C07289=1054.080,253.803,402.120,172.392,36.033,156.770
C07290=1054.086,254.052,402.091,172.395,36.036,156.771
C07291=1054.093,254.300,402.062,172.397,36.039,156.771
C07292=1054.100,254.548,402.034,172.400,36.043,156.772
C07293=1054.106,254.796,402.005,172.402,36.046,156.773
C07294=1054.112,255.044,401.976,172.404,36.050,156.774
C07295=1054.118,255.292,401.947,172.407,36.053,156.774
C07296=1054.125,255.540,401.918,172.410,36.056,156.775
C07297=1054.131,255.789,401.889,172.413,36.060,156.776
C07298=1054.138,256.037,401.859,172.415,36.063,156.777
C07299=1054.144,256.286,401.830,172.417,36.066,156.777
C07300=1054.150,256.534,401.801,172.420,36.070,156.778
C07301=1054.156,256.782,401.772,172.423,36.073,156.779
C07302=1054.163,257.030,401.743,172.425,36.077,156.779
C07303=1054.169,257.278,401.714,172.428,36.081,156.780
C07304=1054.176,257.527,401.685,172.430,36.083,156.781
C07305=1054.183,257.775,401.656,172.433,36.087,156.782
C07306=1054.189,258.023,401.627,172.436,36.091,156.782
C07307=1054.195,258.271,401.598,172.438,36.094,156.783
C07308=1054.201,258.519,401.569,172.441,36.097,156.784
C07309=1054.208,258.768,401.540,172.443,36.101,156.784
C07310=1054.215,259.016,401.511,172.445,36.104,156.785
C07311=1054.221,259.264,401.482,172.449,36.108,156.786
C07312=1054.227,259.512,401.453,172.451,36.111,156.787
C07313=1054.234,259.761,401.423,172.454,36.114,156.787
C07314=1054.241,260.009,401.393,172.456,36.118,156.788
C07315=1054.247,260.257,401.364,172.459,36.121,156.789
C07316=1054.253,260.505,401.335,172.462,36.124,156.789
C07317=1054.260,260.754,401.306,172.464,36.128,156.790
C07318=1054.266,261.002,401.277,172.467,36.131,156.791
C07319=1054.273,261.249,401.247,172.470,36.135,156.792
C07320=1054.279,261.498,401.218,172.472,36.138,156.792
C07321=1054.286,261.746,401.189,172.475,36.141,156.793
C07322=1054.292,261.995,401.160,172.477,36.145,156.794
C07323=1054.298,262.243,401.131,172.481,36.149,156.794
C07324=1054.304,262.456,401.105,172.483,36.151,156.795
C07325=1054.310,262.670,401.079,172.485,36.154,156.796
C07326=1054.316,262.884,401.055,172.487,36.157,156.796
C07327=1054.321,263.098,401.029,172.490,36.160,156.797
C07328=1054.327,263.312,401.003,172.491,36.163,156.798
C07329=1054.332,263.525,400.978,172.494,36.166,156.798
C07330=1054.337,263.740,400.952,172.496,36.169,156.799
C07331=1054.343,263.953,400.927,172.498,36.172,156.799
C07332=1054.351,264.254,400.890,172.502,36.176,156.800
C07333=1054.358,264.554,400.855,172.505,36.180,156.801
C07334=1054.366,264.855,400.819,172.509,36.185,156.802
C07335=1054.373,265.155,400.783,172.511,36.189,156.803
C07336=1054.380,265.403,400.753,172.515,36.192,156.804
C07337=1054.386,265.651,400.724,172.517,36.196,156.804
C07338=1054.392,265.899,400.694,172.519,36.199,156.805
C07339=1054.399,266.148,400.664,172.522,36.203,156.806
C07340=1054.406,266.396,400.635,172.525,36.206,156.807
C07341=1054.411,266.644,400.605,172.528,36.210,156.807
C07342=1054.418,266.892,400.575,172.530,36.213,156.808
C07343=1054.424,267.140,400.546,172.533,36.216,156.809
C07344=1054.431,267.389,400.515,172.536,36.220,156.810
C07345=1054.437,267.636,400.485,172.538,36.223,156.810
C07346=1054.444,267.885,400.456,172.542,36.227,156.811
C07347=1054.450,268.133,400.426,172.544,36.230,156.812
C07348=1054.456,268.381,400.396,172.546,36.234,156.813
C07349=1054.462,268.629,400.366,172.550,36.238,156.813
C07350=1054.469,268.877,400.336,172.552,36.241,156.814
C07351=1054.475,269.126,400.306,172.555,36.245,156.815
C07352=1054.482,269.374,400.276,172.558,36.248,156.816
C07353=1054.488,269.622,400.246,172.560,36.251,156.816
C07354=1054.494,269.869,400.216,172.563,36.255,156.817
C07355=1054.500,270.118,400.186,172.566,36.258,156.818
C07356=1054.507,270.366,400.156,172.569,36.262,156.818
C07357=1054.513,270.614,400.126,172.571,36.265,156.819
C07358=1054.520,270.862,400.096,172.575,36.269,156.820
C07359=1054.526,271.110,400.065,172.577,36.272,156.821
C07360=1054.533,271.359,400.036,172.579,36.276,156.821
C07361=1054.539,271.606,400.006,172.583,36.279,156.822
C07362=1054.546,271.855,399.976,172.585,36.283,156.823
C07363=1054.551,272.102,399.945,172.588,36.286,156.824
C07364=1054.559,272.351,399.915,172.591,36.290,156.825
C07365=1054.564,272.598,399.885,172.594,36.293,156.825
C07366=1054.571,272.847,399.854,172.597,36.297,156.826
C07367=1054.577,273.094,399.824,172.599,36.300,156.827
C07368=1054.584,273.343,399.794,172.602,36.304,156.828
C07369=1054.590,273.591,399.765,172.605,36.307,156.828
C07370=1054.597,273.840,399.734,172.608,36.311,156.829
C07371=1054.602,274.088,399.704,172.610,36.314,156.830
C07372=1054.609,274.336,399.673,172.613,36.318,156.831
C07373=1054.615,274.584,399.643,172.616,36.322,156.831
C07374=1054.622,274.831,399.612,172.619,36.324,156.832
C07375=1054.629,275.079,399.582,172.622,36.328,156.833
C07376=1054.635,275.327,399.551,172.624,36.331,156.833
C07377=1054.641,275.575,399.521,172.628,36.335,156.834
C07378=1054.647,275.824,399.490,172.630,36.339,156.835
C07379=1054.654,276.071,399.460,172.633,36.342,156.836
C07380=1054.660,276.314,399.431,172.636,36.346,156.836
C07381=1054.666,276.555,399.401,172.638,36.349,156.837
C07382=1054.672,276.798,399.371,172.642,36.353,156.838
C07383=1054.679,277.040,399.341,172.644,36.356,156.839
C07384=1054.685,277.282,399.311,172.647,36.360,156.839
C07385=1054.691,277.524,399.281,172.650,36.363,156.840
C07386=1054.697,277.766,399.252,172.652,36.367,156.841
C07387=1054.703,278.007,399.222,172.656,36.370,156.842
C07388=1054.710,278.256,399.192,172.658,36.373,156.842
C07389=1054.716,278.504,399.161,172.661,36.377,156.843
C07390=1054.723,278.751,399.130,172.664,36.381,156.844
C07391=1054.729,279.000,399.099,172.667,36.384,156.845
C07392=1054.735,279.248,399.069,172.670,36.388,156.846
C07393=1054.742,279.496,399.039,172.673,36.391,156.846
C07394=1054.749,279.744,399.007,172.676,36.395,156.847
C07395=1054.755,279.992,398.977,172.678,36.398,156.848
C07396=1054.761,280.240,398.946,172.682,36.402,156.849
C07397=1054.767,280.487,398.915,172.684,36.405,156.849
C07398=1054.774,280.736,398.884,172.688,36.409,156.850
C07399=1054.780,280.984,398.853,172.690,36.412,156.851
C07400=1054.786,281.232,398.822,172.693,36.416,156.852
C07401=1054.793,281.480,398.791,172.696,36.419,156.852
C07402=1054.799,281.728,398.760,172.699,36.423,156.853
C07403=1054.805,281.975,398.729,172.702,36.427,156.854
C07404=1054.812,282.224,398.699,172.704,36.430,156.855
C07405=1054.818,282.472,398.667,172.708,36.434,156.856
C07406=1054.824,282.720,398.637,172.710,36.437,156.856
C07407=1054.831,282.967,398.605,172.714,36.441,156.857
C07408=1054.837,283.216,398.575,172.716,36.444,156.858
C07409=1054.844,283.463,398.544,172.720,36.448,156.859
C07410=1054.850,283.712,398.513,172.722,36.452,156.859
C07411=1054.857,283.960,398.481,172.726,36.455,156.860
C07412=1054.863,284.207,398.451,172.728,36.459,156.861
C07413=1054.869,284.455,398.420,172.732,36.462,156.862
C07414=1054.876,284.703,398.388,172.734,36.466,156.862
C07415=1054.882,284.952,398.357,172.737,36.469,156.863
C07416=1054.889,285.199,398.326,172.740,36.473,156.864
C07417=1054.895,285.447,398.295,172.743,36.477,156.865
C07418=1054.902,285.695,398.264,172.746,36.481,156.866
C07419=1054.908,285.944,398.232,172.749,36.484,156.866
C07420=1054.914,286.191,398.201,172.753,36.488,156.867
C07421=1054.920,286.439,398.170,172.755,36.491,156.868
C07422=1054.927,286.687,398.139,172.759,36.495,156.869
C07423=1054.934,286.935,398.108,172.761,36.498,156.869
C07424=1054.940,287.183,398.076,172.765,36.502,156.870
C07425=1054.946,287.431,398.046,172.767,36.506,156.871
C07426=1054.953,287.679,398.014,172.771,36.509,156.872
C07427=1054.960,287.927,397.983,172.773,36.513,156.873
C07428=1054.966,288.175,397.951,172.776,36.516,156.873
C07429=1054.973,288.422,397.920,172.780,36.520,156.874
C07430=1054.978,288.670,397.888,172.782,36.524,156.875
C07431=1054.985,288.918,397.857,172.786,36.527,156.876
C07432=1054.992,289.166,397.826,172.788,36.531,156.877
C07433=1054.998,289.414,397.795,172.792,36.534,156.877
C07434=1055.004,289.662,397.763,172.794,36.538,156.878
C07435=1055.011,289.910,397.731,172.798,36.542,156.879
C07436=1055.017,290.158,397.700,172.801,36.545,156.880
C07437=1055.024,290.405,397.668,172.804,36.549,156.881
C07438=1055.030,290.652,397.637,172.807,36.553,156.881
C07439=1055.037,290.900,397.606,172.810,36.556,156.882
C07440=1055.042,291.147,397.574,172.813,36.560,156.883
C07441=1055.049,291.395,397.542,172.817,36.563,156.884
C07442=1055.056,291.643,397.510,172.819,36.567,156.885
C07443=1055.062,291.890,397.479,172.823,36.571,156.885
C07444=1055.068,292.138,397.447,172.825,36.574,156.886
C07445=1055.075,292.386,397.416,172.829,36.578,156.887
C07446=1055.082,292.634,397.384,172.832,36.582,156.888
C07447=1055.088,292.882,397.352,172.835,36.585,156.889
C07448=1055.095,293.129,397.320,172.838,36.589,156.889
C07449=1055.101,293.377,397.289,172.842,36.593,156.890
C07450=1055.107,293.625,397.257,172.844,36.596,156.891
C07451=1055.114,293.873,397.225,172.848,36.600,156.892
C07452=1055.120,294.121,397.194,172.850,36.604,156.893
C07453=1055.127,294.368,397.162,172.854,36.607,156.893
C07454=1055.133,294.616,397.130,172.857,36.611,156.894
C07455=1055.139,294.864,397.098,172.860,36.615,156.895
C07456=1055.146,295.112,397.067,172.863,36.618,156.896
C07457=1055.152,295.360,397.034,172.867,36.622,156.897
C07458=1055.159,295.608,397.002,172.869,36.626,156.898
C07459=1055.165,295.856,396.970,172.872,36.629,156.898
C07460=1055.172,296.103,396.938,172.876,36.633,156.899
C07461=1055.178,296.351,396.906,172.879,36.637,156.900
C07462=1055.185,296.599,396.874,172.882,36.640,156.901
C07463=1055.191,296.847,396.842,172.886,36.644,156.902
C07464=1055.197,297.095,396.810,172.888,36.648,156.903
C07465=1055.204,297.342,396.778,172.892,36.652,156.903
C07466=1055.210,297.591,396.746,172.895,36.656,156.904
C07467=1055.216,297.838,396.713,172.898,36.659,156.905
C07468=1055.222,298.086,396.681,172.901,36.663,156.906
C07469=1055.229,298.334,396.648,172.905,36.667,156.907
C07470=1055.236,298.581,396.616,172.907,36.671,156.908
C07471=1055.242,298.829,396.584,172.911,36.674,156.908
C07472=1055.248,299.077,396.551,172.914,36.678,156.909
C07473=1055.254,299.325,396.519,172.917,36.682,156.910
C07474=1055.261,299.573,396.487,172.920,36.686,156.911
C07475=1055.267,299.820,396.455,172.924,36.690,156.912
C07476=1055.273,300.068,396.423,172.926,36.693,156.913
C07477=1055.280,300.316,396.390,172.930,36.697,156.913
C07478=1055.286,300.564,396.357,172.933,36.701,156.914
C07479=1055.293,300.811,396.326,172.937,36.705,156.915
C07480=1055.299,301.059,396.293,172.939,36.709,156.916
C07481=1055.305,301.307,396.260,172.943,36.712,156.917
C07482=1055.311,301.555,396.228,172.946,36.717,156.918
C07483=1055.317,301.802,396.195,172.950,36.720,156.918
C07484=1055.324,302.050,396.163,172.953,36.724,156.919
C07485=1055.331,302.298,396.130,172.956,36.728,156.920
C07486=1055.338,302.546,396.097,172.960,36.731,156.921
C07487=1055.344,302.794,396.065,172.963,36.736,156.922
C07488=1055.350,303.041,396.033,172.966,36.739,156.923
C07489=1055.356,303.289,396.000,172.969,36.743,156.924
C07490=1055.363,303.537,395.967,172.973,36.747,156.924
C07491=1055.370,303.784,395.935,172.976,36.751,156.925
C07492=1055.376,304.047,395.900,172.979,36.755,156.926
C07493=1055.383,304.310,395.866,172.982,36.759,156.927
C07494=1055.390,304.573,395.831,172.986,36.763,156.928
C07495=1055.396,304.836,395.796,172.990,36.767,156.929
C07496=1055.404,305.084,395.764,172.993,36.771,156.930
C07497=1055.410,305.332,395.731,172.997,36.775,156.931
C07498=1055.417,305.580,395.698,173.000,36.778,156.931
C07499=1055.423,305.827,395.666,173.004,36.782,156.932
C07500=1055.429,306.075,395.633,173.006,36.786,156.933
C07501=1055.436,306.323,395.600,173.010,36.790,156.934
C07502=1055.442,306.571,395.567,173.013,36.794,156.935
C07503=1055.449,306.818,395.534,173.017,36.798,156.936
C07504=1055.456,307.065,395.501,173.020,36.801,156.937
C07505=1055.463,307.313,395.468,173.023,36.805,156.938
C07506=1055.469,307.561,395.436,173.027,36.809,156.938
C07507=1055.475,307.808,395.403,173.030,36.813,156.939
C07508=1055.482,308.057,395.370,173.034,36.817,156.940
C07509=1055.489,308.304,395.337,173.037,36.821,156.941
C07510=1055.495,308.552,395.304,173.041,36.825,156.942
C07511=1055.502,308.800,395.271,173.044,36.828,156.943
C07512=1055.508,309.047,395.238,173.047,36.832,156.944
C07513=1055.515,309.294,395.205,173.051,36.836,156.945
C07514=1055.522,309.543,395.172,173.054,36.840,156.945
C07515=1055.529,309.790,395.140,173.058,36.844,156.946
C07516=1055.535,310.037,395.106,173.061,36.848,156.947
C07517=1055.542,310.286,395.073,173.065,36.852,156.948
C07518=1055.548,310.533,395.040,173.068,36.855,156.949
C07519=1055.555,310.781,395.007,173.071,36.859,156.950
C07520=1055.562,311.028,394.974,173.074,36.863,156.951
C07521=1055.569,311.277,394.941,173.078,36.867,156.952
C07522=1055.575,311.524,394.908,173.082,36.871,156.952
C07523=1055.582,311.771,394.874,173.085,36.875,156.953
C07524=1055.589,312.020,394.841,173.089,36.879,156.954
C07525=1055.595,312.267,394.808,173.092,36.883,156.955
C07526=1055.602,312.515,394.775,173.096,36.886,156.956
C07527=1055.608,312.762,394.742,173.099,36.890,156.957
C07528=1055.616,313.010,394.708,173.103,36.894,156.958
C07529=1055.622,313.258,394.675,173.107,36.898,156.959
C07530=1055.629,313.505,394.642,173.109,36.902,156.959
C07531=1055.635,313.753,394.609,173.113,36.906,156.960
C07532=1055.642,314.001,394.574,173.116,36.910,156.961
C07533=1055.648,314.248,394.541,173.120,36.914,156.962
C07534=1055.655,314.497,394.507,173.124,36.918,156.963
C07535=1055.661,314.743,394.474,173.127,36.922,156.964
C07536=1055.667,314.991,394.440,173.131,36.926,156.965
C07537=1055.674,315.239,394.407,173.134,36.930,156.966
C07538=1055.681,315.486,394.373,173.138,36.934,156.967
C07539=1055.687,315.734,394.339,173.142,36.939,156.968
C07540=1055.693,315.982,394.306,173.144,36.943,156.969
C07541=1055.700,316.230,394.272,173.148,36.947,156.970
C07542=1055.706,316.477,394.238,173.151,36.951,156.970
C07543=1055.713,316.725,394.204,173.155,36.955,156.971
C07544=1055.719,316.972,394.171,173.159,36.959,156.972
C07545=1055.726,317.220,394.137,173.162,36.963,156.973
C07546=1055.732,317.467,394.103,173.166,36.967,156.974
C07547=1055.739,317.715,394.069,173.170,36.971,156.975
C07548=1055.745,317.982,394.032,173.173,36.975,156.976
C07549=1055.752,318.249,393.996,173.177,36.980,156.977
C07550=1055.759,318.516,393.959,173.182,36.984,156.978
C07551=1055.767,318.784,393.922,173.185,36.989,156.979
C07552=1055.773,319.031,393.889,173.189,36.993,156.980
C07553=1055.780,319.279,393.854,173.192,36.997,156.981
C07554=1055.786,319.527,393.821,173.196,37.001,156.982
C07555=1055.792,319.774,393.787,173.200,37.005,156.983
C07556=1055.800,320.022,393.753,173.203,37.009,156.984
C07557=1055.805,320.269,393.719,173.207,37.013,156.985
C07558=1055.813,320.517,393.685,173.211,37.017,156.986
C07559=1055.819,320.764,393.650,173.214,37.021,156.987
C07560=1055.826,321.011,393.617,173.218,37.026,156.988
C07561=1055.832,321.259,393.582,173.221,37.030,156.989
C07562=1055.839,321.507,393.548,173.225,37.034,156.990
C07563=1055.845,321.754,393.514,173.229,37.038,156.990
C07564=1055.852,322.002,393.480,173.232,37.042,156.992
C07565=1055.859,322.250,393.446,173.236,37.046,156.992
C07566=1055.866,322.498,393.412,173.240,37.050,156.993
C07567=1055.872,322.745,393.378,173.243,37.054,156.994
C07568=1055.879,322.992,393.343,173.247,37.059,156.995
C07569=1055.885,323.240,393.309,173.251,37.063,156.996
C07570=1055.893,323.488,393.275,173.254,37.067,156.997
C07571=1055.898,323.735,393.241,173.258,37.071,156.998
C07572=1055.906,323.983,393.207,173.262,37.075,156.999
C07573=1055.912,324.230,393.172,173.265,37.079,157.000
C07574=1055.919,324.478,393.138,173.269,37.084,157.001
C07575=1055.926,324.726,393.104,173.272,37.088,157.002
C07576=1055.932,324.972,393.069,173.276,37.092,157.003
C07577=1055.939,325.220,393.035,173.280,37.096,157.004
C07578=1055.946,325.468,393.001,173.284,37.100,157.005
C07579=1055.953,325.715,392.966,173.288,37.105,157.006
C07580=1055.960,325.963,392.932,173.292,37.109,157.007
C07581=1055.966,326.211,392.897,173.295,37.113,157.008
C07582=1055.973,326.458,392.862,173.299,37.117,157.009
C07583=1055.980,326.705,392.829,173.303,37.121,157.010
C07584=1055.987,326.953,392.794,173.306,37.126,157.011
C07585=1055.993,327.201,392.759,173.310,37.130,157.012
C07586=1056.000,327.448,392.725,173.314,37.134,157.013
C07587=1056.007,327.696,392.690,173.318,37.138,157.014
C07588=1056.014,327.943,392.656,173.322,37.142,157.015
C07589=1056.021,328.191,392.621,173.326,37.147,157.016
C07590=1056.028,328.438,392.586,173.329,37.151,157.017
C07591=1056.035,328.686,392.552,173.333,37.155,157.018
C07592=1056.042,328.933,392.517,173.337,37.159,157.019
C07593=1056.048,329.181,392.482,173.341,37.164,157.020
C07594=1056.056,329.428,392.448,173.345,37.168,157.021
C07595=1056.062,329.676,392.413,173.349,37.172,157.022
C07596=1056.069,329.924,392.379,173.353,37.176,157.023
C07597=1056.076,330.171,392.343,173.356,37.181,157.024
C07598=1056.082,330.418,392.308,173.360,37.185,157.025
C07599=1056.089,330.666,392.273,173.364,37.189,157.026
C07600=1056.096,330.914,392.239,173.368,37.194,157.027
C07601=1056.102,331.161,392.204,173.372,37.198,157.028
C07602=1056.109,331.408,392.169,173.376,37.203,157.029
C07603=1056.116,331.656,392.133,173.379,37.207,157.030
C07604=1056.123,331.918,392.097,173.383,37.212,157.031
C07605=1056.130,332.179,392.059,173.388,37.216,157.032
C07606=1056.137,332.441,392.023,173.392,37.221,157.033
C07607=1056.144,332.703,391.985,173.397,37.225,157.034
C07608=1056.151,332.950,391.950,173.400,37.230,157.035
C07609=1056.158,333.198,391.914,173.404,37.234,157.036
C07610=1056.165,333.445,391.879,173.408,37.239,157.037
C07611=1056.172,333.692,391.844,173.411,37.243,157.038
C07612=1056.178,333.940,391.809,173.416,37.248,157.039
C07613=1056.185,334.187,391.774,173.420,37.252,157.040
C07614=1056.192,334.435,391.739,173.424,37.256,157.041
C07615=1056.199,334.682,391.704,173.427,37.261,157.042
C07616=1056.205,334.929,391.669,173.432,37.265,157.043
C07617=1056.213,335.177,391.633,173.436,37.270,157.045
C07618=1056.219,335.425,391.597,173.440,37.274,157.046
C07619=1056.226,335.672,391.562,173.443,37.279,157.047
C07620=1056.233,335.919,391.526,173.448,37.283,157.048
C07621=1056.239,336.167,391.491,173.452,37.288,157.049
C07622=1056.246,336.414,391.456,173.456,37.292,157.050
C07623=1056.254,336.662,391.421,173.459,37.297,157.051
C07624=1056.260,336.909,391.385,173.464,37.301,157.052
C07625=1056.267,337.156,391.349,173.468,37.306,157.053
C07626=1056.273,337.404,391.314,173.472,37.310,157.054
C07627=1056.280,337.651,391.279,173.475,37.315,157.055
C07628=1056.287,337.898,391.242,173.480,37.319,157.056
C07629=1056.294,338.146,391.207,173.484,37.324,157.057
C07630=1056.301,338.393,391.171,173.488,37.329,157.058
C07631=1056.307,338.641,391.135,173.491,37.333,157.060
C07632=1056.314,338.888,391.100,173.496,37.338,157.061
C07633=1056.321,339.135,391.064,173.500,37.342,157.062
C07634=1056.327,339.383,391.028,173.504,37.347,157.063
C07635=1056.335,339.630,390.992,173.509,37.352,157.064
C07636=1056.341,339.877,390.957,173.512,37.356,157.065
C07637=1056.348,340.125,390.920,173.516,37.361,157.066
C07638=1056.355,340.372,390.885,173.521,37.365,157.067
C07639=1056.362,340.619,390.849,173.525,37.370,157.068
C07640=1056.368,340.867,390.814,173.528,37.375,157.069
C07641=1056.376,341.114,390.777,173.533,37.379,157.070
C07642=1056.382,341.361,390.741,173.537,37.384,157.072
C07643=1056.389,341.609,390.706,173.541,37.389,157.073
C07644=1056.397,341.856,390.670,173.546,37.393,157.074
C07645=1056.403,342.103,390.633,173.549,37.398,157.075
C07646=1056.410,342.351,390.598,173.553,37.403,157.076
C07647=1056.417,342.598,390.562,173.558,37.407,157.077
C07648=1056.424,342.845,390.525,173.562,37.412,157.078
C07649=1056.431,343.093,390.490,173.567,37.417,157.079
C07650=1056.437,343.340,390.453,173.570,37.421,157.081
C07651=1056.444,343.587,390.417,173.574,37.426,157.082
C07652=1056.451,343.835,390.381,173.579,37.431,157.083
C07653=1056.458,344.082,390.344,173.583,37.436,157.084
C07654=1056.465,344.329,390.308,173.587,37.440,157.085
C07655=1056.472,344.576,390.272,173.592,37.445,157.086
C07656=1056.479,344.824,390.236,173.595,37.450,157.087
C07657=1056.485,345.071,390.200,173.600,37.455,157.089
C07658=1056.492,345.318,390.163,173.604,37.459,157.090
C07659=1056.499,345.566,390.127,173.608,37.464,157.091
C07660=1056.506,345.823,390.089,173.613,37.469,157.092
C07661=1056.514,346.080,390.051,173.618,37.474,157.093
C07662=1056.520,346.338,390.013,173.622,37.479,157.094
C07663=1056.528,346.596,389.975,173.626,37.484,157.096
C07664=1056.535,346.843,389.939,173.630,37.489,157.097
C07665=1056.542,347.091,389.902,173.635,37.494,157.098
C07666=1056.548,347.337,389.865,173.639,37.499,157.099
C07667=1056.556,347.584,389.829,173.644,37.504,157.100
C07668=1056.563,347.832,389.792,173.648,37.508,157.101
C07669=1056.569,348.079,389.756,173.652,37.513,157.103
C07670=1056.577,348.327,389.719,173.656,37.518,157.104
C07671=1056.584,348.573,389.682,173.660,37.523,157.105
C07672=1056.590,348.821,389.645,173.665,37.528,157.106
C07673=1056.597,349.068,389.609,173.669,37.533,157.107
C07674=1056.605,349.315,389.573,173.674,37.538,157.109
C07675=1056.611,349.562,389.536,173.678,37.543,157.110
C07676=1056.618,349.810,389.499,173.683,37.548,157.111
C07677=1056.625,350.057,389.462,173.687,37.553,157.112
C07678=1056.632,350.303,389.425,173.692,37.558,157.113
C07679=1056.639,350.551,389.389,173.695,37.563,157.115
C07680=1056.647,350.798,389.351,173.700,37.568,157.116
C07681=1056.653,351.045,389.315,173.704,37.572,157.117
C07682=1056.660,351.293,389.278,173.709,37.577,157.118
C07683=1056.668,351.540,389.241,173.713,37.583,157.119
C07684=1056.674,351.787,389.204,173.718,37.588,157.121
C07685=1056.681,352.034,389.167,173.723,37.593,157.122
C07686=1056.689,352.281,389.129,173.727,37.598,157.123
C07687=1056.695,352.528,389.093,173.732,37.603,157.124
C07688=1056.702,352.776,389.055,173.736,37.608,157.126
C07689=1056.709,353.023,389.019,173.740,37.613,157.127
C07690=1056.716,353.270,388.981,173.744,37.618,157.128
C07691=1056.723,353.517,388.944,173.749,37.623,157.129
C07692=1056.730,353.764,388.906,173.753,37.628,157.131
C07693=1056.737,354.012,388.869,173.758,37.633,157.132
C07694=1056.744,354.258,388.832,173.763,37.638,157.133
C07695=1056.751,354.505,388.795,173.767,37.643,157.134
C07696=1056.758,354.752,388.757,173.772,37.649,157.136
C07697=1056.765,355.000,388.720,173.776,37.654,157.137
C07698=1056.772,355.247,388.683,173.781,37.659,157.138
C07699=1056.779,355.494,388.646,173.786,37.664,157.139
C07700=1056.786,355.741,388.608,173.790,37.669,157.141
C07701=1056.794,355.988,388.571,173.795,37.674,157.142
C07702=1056.801,356.235,388.533,173.799,37.680,157.143
C07703=1056.808,356.482,388.496,173.804,37.685,157.144
C07704=1056.815,356.729,388.459,173.809,37.689,157.146
C07705=1056.822,356.976,388.421,173.813,37.695,157.147
C07706=1056.829,357.223,388.383,173.818,37.700,157.148
C07707=1056.837,357.470,388.346,173.823,37.705,157.149
C07708=1056.844,357.717,388.308,173.827,37.710,157.151
C07709=1056.850,357.965,388.270,173.831,37.715,157.152
C07710=1056.858,358.212,388.233,173.837,37.721,157.153
C07711=1056.865,358.459,388.195,173.841,37.726,157.155
C07712=1056.872,358.706,388.158,173.845,37.731,157.156
C07713=1056.879,358.953,388.121,173.851,37.737,157.157
C07714=1056.885,359.200,388.082,173.854,37.742,157.158
C07715=1056.893,359.447,388.044,173.860,37.747,157.160
C07716=1056.900,359.709,388.004,173.865,37.753,157.161
C07717=1056.908,359.971,387.964,173.870,37.759,157.163
C07718=1056.916,360.234,387.924,173.875,37.765,157.164
C07719=1056.923,360.497,387.883,173.880,37.770,157.165
C07720=1056.931,360.744,387.845,173.884,37.776,157.167
C07721=1056.938,360.991,387.808,173.889,37.781,157.168
C07722=1056.945,361.237,387.769,173.894,37.787,157.169
C07723=1056.952,361.485,387.731,173.899,37.791,157.171
C07724=1056.959,361.732,387.694,173.903,37.797,157.172
C07725=1056.967,361.979,387.655,173.908,37.802,157.173
C07726=1056.974,362.226,387.618,173.913,37.808,157.175
C07727=1056.981,362.473,387.579,173.918,37.813,157.176
C07728=1056.988,362.720,387.542,173.922,37.819,157.178
C07729=1056.996,362.966,387.503,173.927,37.824,157.179
C07730=1057.002,363.213,387.465,173.932,37.830,157.180
C07731=1057.010,363.460,387.427,173.937,37.835,157.182
C07732=1057.017,363.707,387.389,173.941,37.841,157.183
C07733=1057.024,363.954,387.351,173.946,37.846,157.184
C07734=1057.030,364.201,387.312,173.952,37.852,157.186
C07735=1057.038,364.447,387.274,173.957,37.857,157.187
C07736=1057.045,364.695,387.234,173.961,37.863,157.188
C07737=1057.053,364.942,387.197,173.966,37.868,157.190
C07738=1057.059,365.189,387.158,173.971,37.874,157.191
C07739=1057.067,365.435,387.120,173.976,37.880,157.193
C07740=1057.074,365.682,387.081,173.981,37.885,157.194
C07741=1057.081,365.929,387.043,173.986,37.891,157.195
C07742=1057.088,366.176,387.004,173.990,37.897,157.197
C07743=1057.095,366.424,386.965,173.995,37.902,157.198
C07744=1057.103,366.670,386.927,174.000,37.908,157.200
C07745=1057.110,366.917,386.888,174.006,37.914,157.201
C07746=1057.117,367.164,386.850,174.011,37.919,157.203
C07747=1057.124,367.410,386.811,174.016,37.925,157.204
C07748=1057.131,367.658,386.772,174.020,37.931,157.205
C07749=1057.139,367.904,386.734,174.025,37.936,157.207
C07750=1057.146,368.151,386.695,174.030,37.942,157.208
C07751=1057.154,368.398,386.656,174.035,37.948,157.210
C07752=1057.161,368.645,386.617,174.041,37.954,157.211
C07753=1057.168,368.892,386.578,174.046,37.959,157.213
C07754=1057.175,369.138,386.540,174.051,37.965,157.214
C07755=1057.183,369.386,386.500,174.056,37.971,157.216
C07756=1057.190,369.632,386.462,174.060,37.977,157.217
C07757=1057.198,369.878,386.423,174.065,37.982,157.218
C07758=1057.205,370.126,386.383,174.070,37.988,157.220
C07759=1057.212,370.372,386.345,174.076,37.994,157.221
C07760=1057.220,370.620,386.306,174.081,38.000,157.223
C07761=1057.227,370.866,386.266,174.086,38.006,157.224
C07762=1057.235,371.113,386.228,174.091,38.012,157.226
C07763=1057.242,371.359,386.188,174.096,38.017,157.227
C07764=1057.249,371.606,386.149,174.101,38.023,157.229
C07765=1057.257,371.854,386.111,174.107,38.029,157.230
C07766=1057.264,372.100,386.071,174.112,38.035,157.232
C07767=1057.272,372.347,386.032,174.117,38.041,157.233
C07768=1057.279,372.593,385.993,174.122,38.047,157.235
C07769=1057.286,372.840,385.954,174.128,38.053,157.236
C07770=1057.293,373.087,385.914,174.133,38.059,157.238
C07771=1057.301,373.333,385.874,174.138,38.065,157.239
C07772=1057.309,373.615,385.830,174.143,38.072,157.241
C07773=1057.317,373.896,385.785,174.150,38.079,157.243
C07774=1057.327,374.177,385.740,174.155,38.086,157.245
C07775=1057.334,374.458,385.695,174.162,38.092,157.246
C07776=1057.342,374.705,385.655,174.167,38.099,157.248
C07777=1057.349,374.951,385.615,174.172,38.105,157.249
C07778=1057.356,375.198,385.576,174.177,38.111,157.251
C07779=1057.364,375.444,385.536,174.183,38.117,157.253
C07780=1057.371,375.691,385.497,174.188,38.123,157.254
C07781=1057.378,375.938,385.457,174.193,38.129,157.256
C07782=1057.386,376.185,385.417,174.198,38.135,157.257
C07783=1057.394,376.431,385.377,174.204,38.141,157.259
C07784=1057.401,376.678,385.338,174.209,38.148,157.260
C07785=1057.408,376.925,385.298,174.214,38.154,157.262
C07786=1057.416,377.172,385.258,174.221,38.160,157.264
C07787=1057.423,377.418,385.218,174.226,38.166,157.265
C07788=1057.431,377.665,385.179,174.231,38.172,157.267
C07789=1057.439,377.912,385.139,174.237,38.179,157.268
C07790=1057.446,378.158,385.099,174.242,38.185,157.270
C07791=1057.454,378.404,385.058,174.247,38.191,157.272
C07792=1057.462,378.651,385.019,174.253,38.198,157.273
C07793=1057.469,378.897,384.979,174.258,38.204,157.275
C07794=1057.476,379.144,384.939,174.263,38.210,157.276
C07795=1057.484,379.391,384.899,174.269,38.216,157.278
C07796=1057.492,379.637,384.858,174.275,38.222,157.280
C07797=1057.499,379.883,384.819,174.280,38.229,157.281
C07798=1057.507,380.130,384.779,174.285,38.235,157.283
C07799=1057.515,380.377,384.739,174.291,38.241,157.284
C07800=1057.523,380.624,384.698,174.296,38.248,157.286
C07801=1057.530,380.870,384.659,174.303,38.254,157.288
C07802=1057.537,381.116,384.618,174.308,38.261,157.290
C07803=1057.545,381.363,384.578,174.313,38.267,157.291
C07804=1057.553,381.609,384.537,174.319,38.274,157.293
C07805=1057.560,381.857,384.497,174.324,38.280,157.295
C07806=1057.568,382.103,384.456,174.331,38.287,157.296
C07807=1057.575,382.349,384.415,174.336,38.293,157.298
C07808=1057.582,382.596,384.375,174.341,38.300,157.300
C07809=1057.590,382.842,384.335,174.347,38.306,157.301
C07810=1057.598,383.089,384.293,174.352,38.313,157.303
C07811=1057.605,383.336,384.253,174.359,38.320,157.305
C07812=1057.613,383.582,384.213,174.364,38.326,157.306
C07813=1057.621,383.828,384.172,174.370,38.333,157.308
C07814=1057.629,384.075,384.131,174.375,38.340,157.310
C07815=1057.636,384.322,384.090,174.381,38.346,157.312
C07816=1057.644,384.568,384.050,174.387,38.353,157.313
C07817=1057.651,384.814,384.009,174.392,38.360,157.315
C07818=1057.658,385.060,383.968,174.399,38.366,157.317
C07819=1057.667,385.307,383.927,174.404,38.373,157.319
C07820=1057.674,385.553,383.887,174.410,38.379,157.320
C07821=1057.682,385.800,383.845,174.416,38.386,157.322
C07822=1057.690,386.047,383.805,174.422,38.393,157.324
C07823=1057.698,386.293,383.764,174.427,38.400,157.326
C07824=1057.706,386.539,383.723,174.434,38.406,157.327
C07825=1057.713,386.786,383.682,174.439,38.413,157.329
C07826=1057.721,387.032,383.641,174.445,38.420,157.331
C07827=1057.729,387.279,383.600,174.451,38.427,157.333
C07828=1057.738,387.591,383.548,174.458,38.435,157.335
C07829=1057.749,387.903,383.496,174.466,38.444,157.337
C07830=1057.759,388.216,383.444,174.473,38.453,157.340
C07831=1057.768,388.529,383.392,174.481,38.462,157.342
C07832=1057.777,388.775,383.350,174.487,38.469,157.344
C07833=1057.784,389.021,383.309,174.493,38.475,157.345
C07834=1057.792,389.267,383.268,174.499,38.482,157.347
C07835=1057.801,389.514,383.227,174.505,38.489,157.349
C07836=1057.808,389.760,383.185,174.511,38.496,157.351
C07837=1057.816,390.006,383.143,174.516,38.503,157.353
C07838=1057.824,390.253,383.103,174.523,38.510,157.355
C07839=1057.832,390.499,383.060,174.529,38.517,157.356
C07840=1057.839,390.746,383.019,174.535,38.524,157.358
C07841=1057.848,390.992,382.978,174.541,38.531,157.360
C07842=1057.855,391.238,382.937,174.547,38.539,157.362
C07843=1057.863,391.485,382.894,174.553,38.546,157.364
C07844=1057.871,391.730,382.853,174.560,38.552,157.366
C07845=1057.879,391.977,382.812,174.565,38.560,157.368
C07846=1057.887,392.224,382.769,174.572,38.567,157.370
C07847=1057.894,392.470,382.728,174.578,38.574,157.372
C07848=1057.903,392.715,382.686,174.584,38.581,157.373
C07849=1057.911,392.962,382.644,174.590,38.589,157.375
C07850=1057.918,393.209,382.603,174.597,38.596,157.377
C07851=1057.926,393.455,382.560,174.602,38.603,157.379
C07852=1057.934,393.701,382.518,174.609,38.610,157.381
C07853=1057.942,393.947,382.476,174.615,38.618,157.383
C07854=1057.951,394.194,382.435,174.621,38.625,157.385
C07855=1057.958,394.440,382.393,174.628,38.632,157.387
C07856=1057.966,394.686,382.350,174.634,38.640,157.389
C07857=1057.974,394.932,382.308,174.641,38.647,157.391
C07858=1057.982,395.179,382.266,174.646,38.654,157.393
C07859=1057.990,395.424,382.224,174.653,38.662,157.395
C07860=1057.998,395.671,382.181,174.660,38.669,157.397
C07861=1058.006,395.917,382.139,174.666,38.677,157.399
C07862=1058.014,396.164,382.097,174.672,38.684,157.401
C07863=1058.022,396.410,382.055,174.679,38.691,157.403
C07864=1058.030,396.656,382.012,174.685,38.699,157.405
C07865=1058.038,396.902,381.970,174.692,38.706,157.407
C07866=1058.047,397.148,381.928,174.697,38.714,157.409
C07867=1058.054,397.394,381.885,174.704,38.722,157.411
C07868=1058.063,397.641,381.842,174.711,38.729,157.413
C07869=1058.070,397.887,381.800,174.717,38.737,157.415
C07870=1058.079,398.133,381.757,174.724,38.745,157.417
C07871=1058.087,398.380,381.715,174.730,38.752,157.419
C07872=1058.095,398.625,381.672,174.737,38.760,157.421
C07873=1058.103,398.871,381.629,174.743,38.767,157.423
C07874=1058.112,399.118,381.587,174.750,38.775,157.425
C07875=1058.119,399.363,381.544,174.757,38.783,157.428
C07876=1058.127,399.610,381.502,174.763,38.791,157.430
C07877=1058.135,399.856,381.459,174.770,38.799,157.432
C07878=1058.144,400.102,381.415,174.777,38.807,157.434
C07879=1058.152,400.348,381.372,174.783,38.814,157.436
C07880=1058.160,400.594,381.331,174.790,38.822,157.438
C07881=1058.168,400.840,381.287,174.796,38.830,157.440
C07882=1058.176,401.087,381.244,174.803,38.838,157.442
C07883=1058.185,401.333,381.201,174.810,38.846,157.445
C07884=1058.196,401.663,381.144,174.819,38.856,157.447
C07885=1058.207,401.992,381.086,174.828,38.867,157.450
C07886=1058.218,402.323,381.028,174.837,38.877,157.453
C07887=1058.229,402.652,380.970,174.846,38.888,157.456
C07888=1058.237,402.898,380.926,174.853,38.896,157.458
C07889=1058.245,403.144,380.883,174.860,38.904,157.460
C07890=1058.254,403.390,380.840,174.866,38.912,157.463
C07891=1058.262,403.637,380.797,174.873,38.920,157.465
C07892=1058.270,403.882,380.753,174.881,38.929,157.467
C07893=1058.279,404.128,380.710,174.887,38.936,157.469
C07894=1058.287,404.374,380.666,174.895,38.945,157.472
C07895=1058.295,404.621,380.623,174.902,38.953,157.474
C07896=1058.304,404.867,380.579,174.909,38.961,157.476
C07897=1058.312,405.113,380.536,174.916,38.969,157.478
C07898=1058.320,405.359,380.491,174.923,38.977,157.481
C07899=1058.329,405.605,380.448,174.930,38.986,157.483
C07900=1058.337,405.851,380.405,174.937,38.994,157.485
C07901=1058.345,406.097,380.361,174.944,39.003,157.487
C07902=1058.354,406.342,380.317,174.951,39.011,157.490
C07903=1058.361,406.589,380.273,174.958,39.019,157.492
C07904=1058.371,406.835,380.229,174.965,39.027,157.494
C07905=1058.378,407.081,380.185,174.972,39.036,157.497
C07906=1058.387,407.327,380.141,174.980,39.045,157.499
C07907=1058.395,407.572,380.097,174.987,39.053,157.501
C07908=1058.404,407.819,380.052,174.994,39.061,157.504
C07909=1058.413,408.065,380.009,175.001,39.070,157.506
C07910=1058.421,408.311,379.965,175.008,39.078,157.508
C07911=1058.429,408.556,379.921,175.016,39.087,157.511
C07912=1058.438,408.803,379.877,175.023,39.095,157.513
C07913=1058.446,409.048,379.832,175.030,39.104,157.515
C07914=1058.454,409.294,379.788,175.037,39.113,157.518
C07915=1058.464,409.540,379.744,175.045,39.121,157.520
C07916=1058.472,409.786,379.700,175.053,39.130,157.523
C07917=1058.480,410.032,379.655,175.060,39.139,157.525
C07918=1058.489,410.278,379.611,175.067,39.147,157.527
C07919=1058.498,410.524,379.566,175.074,39.156,157.530
C07920=1058.506,410.770,379.522,175.083,39.165,157.532
C07921=1058.514,411.015,379.477,175.090,39.173,157.535
C07922=1058.524,411.261,379.433,175.097,39.182,157.537
C07923=1058.532,411.508,379.388,175.105,39.191,157.540
C07924=1058.540,411.753,379.344,175.112,39.200,157.542
C07925=1058.550,411.999,379.299,175.120,39.209,157.545
C07926=1058.558,412.245,379.255,175.128,39.218,157.547
C07927=1058.567,412.491,379.210,175.135,39.227,157.550
C07928=1058.575,412.736,379.165,175.143,39.235,157.552
C07929=1058.585,412.982,379.121,175.151,39.244,157.555
C07930=1058.594,413.228,379.075,175.158,39.254,157.557
C07931=1058.602,413.474,379.031,175.166,39.262,157.560
C07932=1058.611,413.720,378.986,175.174,39.271,157.562
C07933=1058.619,413.966,378.941,175.181,39.281,157.565
C07934=1058.628,414.212,378.896,175.190,39.289,157.567
C07935=1058.637,414.457,378.850,175.197,39.299,157.570
C07936=1058.646,414.703,378.805,175.205,39.308,157.573
C07937=1058.655,414.949,378.760,175.213,39.317,157.575
C07938=1058.663,415.195,378.715,175.221,39.326,157.578
C07939=1058.672,415.440,378.670,175.229,39.336,157.580
C07940=1058.679,415.655,378.630,175.235,39.344,157.583
C07941=1058.687,415.870,378.591,175.242,39.352,157.585
C07942=1058.696,416.085,378.551,175.250,39.360,157.587
C07943=1058.703,416.300,378.511,175.257,39.368,157.590
C07944=1058.710,416.515,378.471,175.264,39.376,157.592
C07945=1058.719,416.729,378.432,175.270,39.384,157.594
C07946=1058.726,416.944,378.392,175.278,39.393,157.597
C07947=1058.734,417.159,378.352,175.285,39.401,157.599
C07948=1058.743,417.405,378.307,175.293,39.410,157.602
C07949=1058.752,417.651,378.261,175.301,39.420,157.604
C07950=1058.761,417.897,378.216,175.310,39.429,157.607
C07951=1058.770,418.142,378.170,175.317,39.439,157.610
C07952=1058.779,418.388,378.124,175.326,39.448,157.613
C07953=1058.787,418.634,378.078,175.334,39.458,157.615
C07954=1058.796,418.879,378.032,175.342,39.467,157.618
C07955=1058.805,419.125,377.987,175.351,39.477,157.621
C07956=1058.815,419.370,377.940,175.359,39.487,157.624
C07957=1058.824,419.616,377.895,175.367,39.496,157.626
C07958=1058.834,419.862,377.849,175.376,39.506,157.629
C07959=1058.842,420.108,377.803,175.384,39.516,157.632
C07960=1058.851,420.353,377.756,175.393,39.526,157.635
C07961=1058.860,420.598,377.710,175.401,39.535,157.638
C07962=1058.869,420.844,377.664,175.410,39.545,157.640
C07963=1058.878,421.090,377.618,175.418,39.555,157.643
C07964=1058.887,421.335,377.572,175.427,39.565,157.646
C07965=1058.896,421.580,377.525,175.435,39.575,157.649
C07966=1058.906,421.826,377.479,175.444,39.585,157.652
C07967=1058.915,422.071,377.433,175.452,39.595,157.655
C07968=1058.923,422.317,377.386,175.461,39.605,157.658
C07969=1058.933,422.562,377.340,175.470,39.615,157.661
C07970=1058.942,422.808,377.293,175.479,39.625,157.663
C07971=1058.951,423.054,377.247,175.488,39.635,157.666
C07972=1058.960,423.299,377.200,175.497,39.645,157.669
C07973=1058.970,423.545,377.153,175.504,39.656,157.672
C07974=1058.979,423.790,377.106,175.513,39.666,157.675
C07975=1058.988,424.035,377.060,175.522,39.676,157.678
C07976=1058.998,424.281,377.013,175.531,39.686,157.681
C07977=1059.006,424.527,376.966,175.540,39.697,157.684
C07978=1059.016,424.772,376.919,175.549,39.707,157.687
C07979=1059.025,425.017,376.873,175.558,39.717,157.690
C07980=1059.034,425.262,376.826,175.567,39.727,157.693
C07981=1059.044,425.508,376.779,175.576,39.737,157.696
C07982=1059.053,425.753,376.732,175.585,39.748,157.699
C07983=1059.063,425.999,376.685,175.594,39.758,157.702
C07984=1059.072,426.244,376.637,175.604,39.769,157.706
C07985=1059.081,426.489,376.590,175.613,39.779,157.709
C07986=1059.091,426.735,376.543,175.622,39.790,157.712
C07987=1059.100,426.980,376.496,175.632,39.801,157.715
C07988=1059.116,427.376,376.419,175.646,39.818,157.720
C07989=1059.131,427.773,376.342,175.661,39.835,157.725
C07990=1059.146,428.168,376.266,175.676,39.853,157.730
C07991=1059.161,428.565,376.189,175.691,39.870,157.735
C07992=1059.171,428.810,376.142,175.702,39.880,157.739
C07993=1059.181,429.055,376.094,175.711,39.892,157.742
C07994=1059.190,429.300,376.045,175.720,39.902,157.745
C07995=1059.200,429.545,375.999,175.730,39.913,157.748
C07996=1059.214,429.902,375.929,175.744,39.929,157.753
C07997=1059.228,430.259,375.859,175.758,39.945,157.758
C07998=1059.242,430.615,375.789,175.772,39.961,157.763
C07999=1059.256,430.971,375.719,175.786,39.977,157.767
C08000=1059.265,431.217,375.672,175.797,39.989,157.771
C08001=1059.275,431.462,375.623,175.806,40.000,157.774
C08002=1059.285,431.707,375.575,175.815,40.011,157.778
C08003=1059.295,431.952,375.526,175.826,40.022,157.781
C08004=1059.304,432.197,375.478,175.835,40.034,157.784
C08005=1059.314,432.442,375.430,175.846,40.045,157.788
C08006=1059.324,432.687,375.381,175.856,40.056,157.791
C08007=1059.333,432.932,375.333,175.866,40.067,157.795
C08008=1059.343,433.177,375.284,175.876,40.079,157.798
C08009=1059.353,433.422,375.236,175.886,40.091,157.802
C08010=1059.363,433.667,375.187,175.896,40.102,157.805
C08011=1059.372,433.912,375.139,175.906,40.114,157.809
C08012=1059.382,434.157,375.090,175.917,40.125,157.812
C08013=1059.393,434.403,375.041,175.927,40.137,157.816
C08014=1059.403,434.647,374.992,175.937,40.148,157.819
C08015=1059.412,434.892,374.943,175.948,40.160,157.823
C08016=1059.422,435.137,374.895,175.958,40.172,157.826
C08017=1059.433,435.382,374.845,175.969,40.184,157.830
C08018=1059.443,435.627,374.797,175.979,40.195,157.833
C08019=1059.453,435.871,374.747,175.990,40.207,157.837
C08020=1059.463,436.117,374.699,176.000,40.219,157.841
C08021=1059.473,436.361,374.649,176.011,40.231,157.844
C08022=1059.482,436.607,374.600,176.021,40.243,157.848
C08023=1059.493,436.852,374.551,176.032,40.255,157.852
C08024=1059.503,437.096,374.501,176.043,40.267,157.855
C08025=1059.513,437.342,374.452,176.053,40.279,157.859
C08026=1059.523,437.586,374.403,176.064,40.291,157.863
C08027=1059.534,437.831,374.354,176.075,40.303,157.866
C08028=1059.543,438.076,374.304,176.086,40.315,157.870
C08029=1059.554,438.321,374.254,176.097,40.327,157.874
C08030=1059.564,438.565,374.205,176.108,40.339,157.878
C08031=1059.575,438.810,374.155,176.119,40.351,157.881
C08032=1059.584,439.055,374.105,176.130,40.364,157.885
C08033=1059.595,439.299,374.055,176.141,40.376,157.889
C08034=1059.606,439.545,374.006,176.152,40.389,157.893
C08035=1059.615,439.789,373.956,176.163,40.401,157.897
C08036=1059.626,440.034,373.906,176.174,40.414,157.901
C08037=1059.637,440.279,373.856,176.185,40.426,157.905
C08038=1059.646,440.523,373.806,176.198,40.439,157.909
C08039=1059.657,440.768,373.756,176.209,40.451,157.912
C08040=1059.667,441.013,373.705,176.220,40.464,157.916
C08041=1059.678,441.258,373.655,176.231,40.477,157.920
C08042=1059.689,441.502,373.605,176.243,40.490,157.924
C08043=1059.698,441.746,373.554,176.255,40.502,157.928
C08044=1059.709,441.991,373.505,176.266,40.515,157.932
C08045=1059.719,442.236,373.454,176.278,40.528,157.936
C08046=1059.730,442.480,373.403,176.289,40.540,157.940
C08047=1059.741,442.725,373.352,176.301,40.553,157.944
C08048=1059.751,442.969,373.302,176.313,40.567,157.949
C08049=1059.762,443.214,373.251,176.324,40.579,157.953
C08050=1059.773,443.459,373.201,176.337,40.592,157.957
C08051=1059.783,443.703,373.150,176.348,40.606,157.961
C08052=1059.799,444.048,373.078,176.366,40.624,157.967
C08053=1059.813,444.392,373.006,176.382,40.642,157.973
C08054=1059.828,444.737,372.935,176.399,40.661,157.979
C08055=1059.843,445.082,372.862,176.417,40.680,157.985
C08056=1059.854,445.326,372.811,176.429,40.694,157.989
C08057=1059.865,445.571,372.760,176.441,40.707,157.993
C08058=1059.876,445.816,372.708,176.454,40.720,157.998
C08059=1059.887,446.059,372.657,176.466,40.734,158.002
C08060=1059.898,446.304,372.606,176.479,40.747,158.006
C08061=1059.908,446.549,372.554,176.491,40.761,158.010
C08062=1059.920,446.793,372.503,176.503,40.774,158.015
C08063=1059.930,447.037,372.452,176.516,40.788,158.019
C08064=1059.942,447.280,372.400,176.529,40.802,158.024
C08065=1059.955,447.523,372.350,176.542,40.815,158.028
C08066=1059.966,447.767,372.300,176.554,40.828,158.032
C08067=1059.981,448.012,372.250,176.567,40.841,158.036
C08068=1059.996,448.256,372.202,176.581,40.853,158.041
C08069=1060.011,448.500,372.154,176.593,40.866,158.045
C08070=1060.028,448.745,372.107,176.606,40.878,158.049
C08071=1060.046,448.990,372.059,176.620,40.890,158.053
C08072=1060.064,449.234,372.013,176.632,40.902,158.057
C08073=1060.083,449.480,371.967,176.646,40.913,158.060
C08074=1060.103,449.725,371.922,176.660,40.924,158.064
C08075=1060.124,449.970,371.879,176.673,40.935,158.068
C08076=1059.794,449.982,371.599,176.668,41.048,158.099
C08077=1059.773,449.738,371.644,176.654,41.037,158.095
C08078=1059.752,449.492,371.688,176.641,41.026,158.092
C08079=1059.733,449.247,371.734,176.628,41.014,158.088
C08080=1059.714,449.001,371.781,176.614,41.003,158.084
C08081=1059.697,448.756,371.827,176.601,40.991,158.080
C08082=1059.680,448.512,371.875,176.587,40.979,158.076
C08083=1059.664,448.268,371.923,176.575,40.966,158.072
C08084=1059.649,448.024,371.971,176.561,40.954,158.067
C08085=1059.635,447.779,372.021,176.548,40.941,158.063
C08086=1059.621,447.535,372.071,176.536,40.928,158.059
C08087=1059.609,447.291,372.121,176.523,40.915,158.055
C08088=1059.598,447.049,372.172,176.510,40.902,158.050
C08089=1059.587,446.804,372.224,176.497,40.888,158.046
C08090=1059.576,446.560,372.276,176.484,40.875,158.042
C08091=1059.565,446.316,372.326,176.472,40.861,158.037
C08092=1059.554,446.071,372.378,176.459,40.847,158.033
C08093=1059.543,445.827,372.430,176.447,40.834,158.029
C08094=1059.532,445.583,372.481,176.434,40.821,158.024
C08095=1059.522,445.338,372.532,176.422,40.807,158.020
C08096=1059.510,445.094,372.583,176.409,40.794,158.016
C08097=1059.496,444.768,372.651,176.393,40.776,158.010
C08098=1059.482,444.443,372.720,176.377,40.759,158.004
C08099=1059.468,444.117,372.787,176.361,40.742,157.999
C08100=1059.454,443.792,372.855,176.345,40.724,157.993
C08101=1059.443,443.548,372.905,176.333,40.711,157.989
C08102=1059.432,443.304,372.957,176.321,40.698,157.985
C08103=1059.421,443.059,373.007,176.309,40.685,157.981
C08104=1059.411,442.814,373.058,176.297,40.672,157.977
C08105=1059.400,442.570,373.108,176.285,40.659,157.972
C08106=1059.390,442.325,373.159,176.274,40.646,157.968
C08107=1059.379,442.081,373.210,176.261,40.634,157.964
C08108=1059.368,441.836,373.261,176.250,40.621,157.960
C08109=1059.358,441.591,373.310,176.239,40.608,157.956
C08110=1059.347,441.346,373.361,176.226,40.595,157.952
C08111=1059.337,441.102,373.411,176.215,40.583,157.948
C08112=1059.326,440.858,373.461,176.204,40.570,157.944
C08113=1059.316,440.613,373.512,176.192,40.558,157.940
C08114=1059.305,440.368,373.562,176.181,40.545,157.937
C08115=1059.295,440.123,373.612,176.169,40.533,157.933
C08116=1059.285,439.879,373.662,176.158,40.520,157.929
C08117=1059.274,439.634,373.712,176.147,40.508,157.925
C08118=1059.264,439.389,373.762,176.136,40.496,157.921
C08119=1059.253,439.144,373.812,176.124,40.483,157.917
C08120=1059.243,438.900,373.861,176.113,40.471,157.913
C08121=1059.233,438.655,373.912,176.102,40.458,157.909
C08122=1059.223,438.410,373.961,176.091,40.446,157.906
C08123=1059.213,438.165,374.011,176.080,40.434,157.902
C08124=1059.203,437.921,374.060,176.069,40.422,157.898
C08125=1059.193,437.675,374.110,176.058,40.410,157.894
C08126=1059.183,437.431,374.159,176.047,40.398,157.891
C08127=1059.172,437.186,374.209,176.036,40.386,157.887
C08128=1059.161,436.941,374.258,176.025,40.374,157.883
C08129=1059.151,436.696,374.307,176.015,40.362,157.880
C08130=1059.141,436.451,374.357,176.004,40.350,157.876
C08131=1059.131,436.207,374.406,175.993,40.338,157.872
C08132=1059.121,435.962,374.454,175.983,40.327,157.869
C08133=1059.110,435.717,374.504,175.972,40.315,157.865
C08134=1059.101,435.471,374.553,175.962,40.303,157.861
C08135=1059.091,435.227,374.602,175.951,40.291,157.858
C08136=1059.081,434.981,374.651,175.940,40.280,157.854
C08137=1059.071,434.737,374.700,175.930,40.268,157.851
C08138=1059.061,434.492,374.749,175.920,40.257,157.847
C08139=1059.051,434.247,374.798,175.909,40.245,157.844
C08140=1059.041,434.001,374.846,175.899,40.234,157.840
C08141=1059.031,433.757,374.896,175.889,40.222,157.837
C08142=1059.021,433.512,374.944,175.878,40.210,157.833
C08143=1059.011,433.267,374.993,175.869,40.199,157.830
C08144=1059.002,433.022,375.041,175.858,40.188,157.826
C08145=1058.992,432.777,375.090,175.848,40.176,157.823
C08146=1058.982,432.532,375.138,175.838,40.165,157.819
C08147=1058.972,432.287,375.187,175.828,40.154,157.816
C08148=1058.963,432.042,375.235,175.818,40.142,157.812
C08149=1058.953,431.797,375.283,175.808,40.131,157.809
C08150=1058.943,431.552,375.332,175.798,40.120,157.806
C08151=1058.934,431.307,375.380,175.788,40.109,157.802
C08152=1058.923,431.062,375.428,175.778,40.098,157.799
C08153=1058.910,430.703,375.498,175.764,40.081,157.794
C08154=1058.895,430.344,375.569,175.750,40.065,157.789
C08155=1058.881,429.987,375.639,175.735,40.049,157.784
C08156=1058.866,429.627,375.709,175.721,40.033,157.779
C08157=1058.858,429.382,375.756,175.711,40.022,157.776
C08158=1058.848,429.138,375.805,175.701,40.011,157.773
C08159=1058.838,428.892,375.853,175.692,40.001,157.770
C08160=1058.828,428.647,375.900,175.682,39.990,157.767
C08161=1058.819,428.402,375.947,175.673,39.979,157.763
C08162=1058.810,428.156,375.995,175.664,39.968,157.760
C08163=1058.799,427.911,376.043,175.653,39.957,157.757
C08164=1058.790,427.666,376.091,175.644,39.947,157.754
C08165=1058.781,427.421,376.138,175.635,39.936,157.751
C08166=1058.772,427.175,376.185,175.626,39.926,157.747
C08167=1058.762,426.930,376.232,175.617,39.915,157.744
C08168=1058.753,426.685,376.280,175.607,39.904,157.741
C08169=1058.743,426.439,376.328,175.597,39.894,157.738
C08170=1058.734,426.194,376.375,175.588,39.884,157.735
C08171=1058.725,425.948,376.422,175.579,39.873,157.732
C08172=1058.714,425.703,376.469,175.570,39.863,157.729
C08173=1058.706,425.458,376.516,175.561,39.853,157.726
C08174=1058.696,425.212,376.563,175.552,39.842,157.723
C08175=1058.686,424.968,376.610,175.543,39.832,157.720
C08176=1058.677,424.721,376.657,175.534,39.821,157.717
C08177=1058.667,424.477,376.704,175.525,39.811,157.714
C08178=1058.659,424.231,376.750,175.516,39.801,157.711
C08179=1058.649,423.985,376.797,175.507,39.791,157.708
C08180=1058.640,423.740,376.844,175.498,39.781,157.705
C08181=1058.630,423.495,376.891,175.489,39.770,157.702
C08182=1058.621,423.249,376.937,175.480,39.760,157.699
C08183=1058.612,423.004,376.984,175.472,39.750,157.696
C08184=1058.602,422.758,377.030,175.463,39.740,157.693
C08185=1058.594,422.513,377.078,175.454,39.730,157.690
C08186=1058.584,422.268,377.124,175.445,39.720,157.687
C08187=1058.574,422.022,377.170,175.436,39.711,157.684
C08188=1058.566,421.776,377.217,175.427,39.700,157.681
C08189=1058.557,421.531,377.263,175.419,39.690,157.678
C08190=1058.548,421.286,377.310,175.410,39.681,157.675
C08191=1058.539,421.040,377.355,175.402,39.670,157.672
C08192=1058.530,420.795,377.401,175.393,39.661,157.670
C08193=1058.521,420.548,377.449,175.385,39.651,157.667
C08194=1058.511,420.303,377.495,175.376,39.641,157.664
C08195=1058.502,420.058,377.541,175.367,39.631,157.661
C08196=1058.494,419.812,377.587,175.359,39.622,157.658
C08197=1058.485,419.567,377.633,175.351,39.612,157.656
C08198=1058.476,419.321,377.678,175.342,39.603,157.653
C08199=1058.466,419.076,377.725,175.333,39.593,157.650
C08200=1058.457,418.830,377.770,175.326,39.584,157.647
C08201=1058.445,418.502,377.831,175.314,39.571,157.644
C08202=1058.433,418.175,377.892,175.303,39.558,157.640
C08203=1058.421,417.849,377.953,175.292,39.545,157.636
C08204=1058.409,417.521,378.014,175.281,39.533,157.633
C08205=1058.400,417.275,378.059,175.273,39.523,157.630
C08206=1058.391,417.030,378.106,175.265,39.514,157.627
C08207=1058.383,416.785,378.151,175.257,39.505,157.625
C08208=1058.374,416.539,378.196,175.249,39.495,157.622
C08209=1058.364,416.283,378.243,175.240,39.485,157.619
C08210=1058.355,416.027,378.290,175.231,39.476,157.616
C08211=1058.346,415.771,378.338,175.224,39.466,157.614
C08212=1058.336,415.516,378.385,175.215,39.456,157.611
C08213=1058.328,415.269,378.430,175.207,39.447,157.608
C08214=1058.319,415.024,378.476,175.199,39.438,157.606
C08215=1058.310,414.778,378.521,175.192,39.429,157.603
C08216=1058.301,414.533,378.566,175.183,39.420,157.600
C08217=1058.293,414.286,378.612,175.176,39.411,157.598
C08218=1058.285,414.041,378.657,175.167,39.402,157.595
C08219=1058.276,413.795,378.702,175.160,39.393,157.593
C08220=1058.266,413.549,378.747,175.152,39.383,157.590
C08221=1058.257,413.304,378.792,175.144,39.375,157.588
C08222=1058.249,413.058,378.836,175.136,39.366,157.585
C08223=1058.240,412.812,378.882,175.129,39.357,157.583
C08224=1058.231,412.566,378.926,175.121,39.348,157.580
C08225=1058.222,412.321,378.971,175.113,39.339,157.578
C08226=1058.214,412.074,379.016,175.106,39.330,157.575
C08227=1058.204,411.828,379.060,175.097,39.322,157.573
C08228=1058.196,411.583,379.105,175.090,39.313,157.570
C08229=1058.187,411.337,379.149,175.083,39.304,157.568
C08230=1058.179,411.091,379.194,175.075,39.295,157.565
C08231=1058.170,410.845,379.238,175.067,39.286,157.563
C08232=1058.161,410.600,379.283,175.060,39.278,157.560
C08233=1058.153,410.353,379.328,175.052,39.269,157.558
C08234=1058.144,410.108,379.371,175.045,39.260,157.555
C08235=1058.135,409.861,379.416,175.038,39.252,157.553
C08236=1058.127,409.615,379.460,175.029,39.243,157.551
C08237=1058.118,409.370,379.504,175.022,39.234,157.548
C08238=1058.110,409.124,379.549,175.015,39.226,157.546
C08239=1058.102,408.878,379.593,175.008,39.217,157.543
C08240=1058.092,408.632,379.637,175.001,39.209,157.541
C08241=1058.084,408.386,379.682,174.993,39.200,157.539
C08242=1058.076,408.140,379.726,174.986,39.192,157.536
C08243=1058.067,407.894,379.770,174.979,39.183,157.534
C08244=1058.059,407.648,379.814,174.972,39.175,157.532
C08245=1058.051,407.402,379.858,174.964,39.166,157.529
C08246=1058.042,407.157,379.902,174.956,39.158,157.527
C08247=1058.033,406.910,379.947,174.949,39.149,157.524
C08248=1058.025,406.664,379.990,174.942,39.141,157.522
C08249=1058.017,406.418,380.034,174.935,39.133,157.520
C08250=1058.009,406.173,380.078,174.928,39.125,157.518
C08251=1058.000,405.927,380.121,174.920,39.116,157.515
C08252=1057.992,405.681,380.166,174.913,39.108,157.513
C08253=1057.983,405.434,380.209,174.906,39.099,157.511
C08254=1057.975,405.188,380.253,174.899,39.092,157.508
C08255=1057.967,404.942,380.296,174.893,39.083,157.506
C08256=1057.958,404.696,380.341,174.886,39.075,157.504
C08257=1057.950,404.450,380.384,174.879,39.067,157.502
C08258=1057.942,404.204,380.427,174.872,39.058,157.499
C08259=1057.933,403.959,380.471,174.865,39.050,157.497
C08260=1057.926,403.712,380.515,174.858,39.043,157.495
C08261=1057.917,403.466,380.558,174.851,39.034,157.493
C08262=1057.909,403.220,380.601,174.844,39.026,157.490
C08263=1057.901,402.974,380.644,174.837,39.018,157.488
C08264=1057.892,402.728,380.688,174.830,39.011,157.486
C08265=1057.880,402.396,380.747,174.821,38.999,157.483
C08266=1057.869,402.065,380.805,174.811,38.989,157.480
C08267=1057.858,401.732,380.862,174.802,38.978,157.477
C08268=1057.847,401.401,380.920,174.793,38.968,157.474
C08269=1057.839,401.154,380.964,174.786,38.960,157.472
C08270=1057.831,400.908,381.007,174.780,38.952,157.470
C08271=1057.822,400.662,381.050,174.773,38.944,157.468
C08272=1057.814,400.417,381.093,174.766,38.936,157.466
C08273=1057.806,400.170,381.135,174.759,38.929,157.464
C08274=1057.798,399.924,381.178,174.752,38.921,157.462
C08275=1057.790,399.678,381.222,174.746,38.913,157.459
C08276=1057.781,399.432,381.265,174.739,38.905,157.457
C08277=1057.774,399.186,381.307,174.732,38.898,157.455
C08278=1057.765,398.940,381.350,174.726,38.890,157.453
C08279=1057.757,398.694,381.393,174.720,38.882,157.451
C08280=1057.749,398.447,381.435,174.713,38.875,157.449
C08281=1057.741,398.202,381.478,174.706,38.867,157.447
C08282=1057.733,397.955,381.520,174.700,38.859,157.445
C08283=1057.725,397.709,381.564,174.693,38.852,157.443
C08284=1057.717,397.463,381.606,174.686,38.844,157.441
C08285=1057.709,397.217,381.649,174.681,38.837,157.439
C08286=1057.700,396.970,381.691,174.674,38.829,157.437
C08287=1057.693,396.724,381.733,174.667,38.822,157.435
C08288=1057.684,396.478,381.776,174.661,38.814,157.433
C08289=1057.676,396.231,381.818,174.654,38.807,157.431
C08290=1057.669,395.985,381.860,174.648,38.800,157.429
C08291=1057.660,395.739,381.902,174.642,38.792,157.427
C08292=1057.652,395.494,381.944,174.635,38.785,157.425
C08293=1057.644,395.247,381.987,174.628,38.777,157.423
C08294=1057.636,395.001,382.029,174.622,38.770,157.421
C08295=1057.628,394.754,382.071,174.616,38.762,157.419
C08296=1057.620,394.508,382.113,174.610,38.755,157.417
C08297=1057.612,394.262,382.155,174.603,38.748,157.415
C08298=1057.604,394.016,382.197,174.596,38.741,157.413
C08299=1057.596,393.769,382.240,174.591,38.733,157.411
C08300=1057.588,393.523,382.281,174.584,38.726,157.409
C08301=1057.580,393.277,382.323,174.578,38.719,157.407
C08302=1057.572,393.031,382.365,174.571,38.711,157.405
C08303=1057.564,392.785,382.407,174.566,38.704,157.403
C08304=1057.556,392.538,382.449,174.559,38.697,157.401
C08305=1057.548,392.292,382.490,174.553,38.690,157.399
C08306=1057.541,392.046,382.532,174.547,38.682,157.397
C08307=1057.532,391.799,382.574,174.541,38.675,157.396
C08308=1057.525,391.553,382.616,174.534,38.669,157.394
C08309=1057.517,391.307,382.657,174.529,38.662,157.392
C08310=1057.509,391.060,382.699,174.522,38.654,157.390
C08311=1057.501,390.814,382.741,174.516,38.647,157.388
C08312=1057.493,390.568,382.782,174.510,38.640,157.386
C08313=1057.485,390.321,382.824,174.504,38.633,157.384
C08314=1057.478,390.075,382.865,174.498,38.626,157.382
C08315=1057.469,389.829,382.907,174.492,38.619,157.380
C08316=1057.462,389.582,382.948,174.485,38.612,157.379
C08317=1057.453,389.336,382.990,174.480,38.606,157.377
C08318=1057.446,389.089,383.031,174.474,38.599,157.375
C08319=1057.437,388.844,383.072,174.468,38.592,157.373
C08320=1057.430,388.597,383.113,174.462,38.585,157.371
C08321=1057.420,388.283,383.166,174.454,38.576,157.369
C08322=1057.410,387.969,383.218,174.446,38.567,157.367
C08323=1057.400,387.654,383.271,174.439,38.558,157.364
C08324=1057.390,387.340,383.324,174.431,38.550,157.362
C08325=1057.382,387.094,383.364,174.425,38.543,157.360
C08326=1057.374,386.847,383.405,174.419,38.537,157.359
C08327=1057.366,386.601,383.446,174.413,38.530,157.357
C08328=1057.359,386.354,383.487,174.408,38.523,157.355
C08329=1057.350,386.107,383.528,174.401,38.516,157.353
C08330=1057.342,385.861,383.569,174.396,38.509,157.351
C08331=1057.335,385.615,383.610,174.390,38.503,157.350
C08332=1057.327,385.368,383.651,174.384,38.496,157.348
C08333=1057.320,385.122,383.692,174.378,38.489,157.346
C08334=1057.312,384.875,383.733,174.373,38.483,157.345
C08335=1057.304,384.629,383.773,174.367,38.476,157.343
C08336=1057.296,384.382,383.815,174.361,38.469,157.341
C08337=1057.288,384.136,383.855,174.355,38.463,157.339
C08338=1057.281,383.890,383.896,174.350,38.456,157.338
C08339=1057.273,383.643,383.936,174.343,38.449,157.336
C08340=1057.266,383.397,383.977,174.338,38.443,157.334
C08341=1057.259,383.151,384.018,174.332,38.437,157.332
C08342=1057.251,382.904,384.058,174.327,38.430,157.331
C08343=1057.243,382.657,384.098,174.322,38.424,157.329
C08344=1057.236,382.411,384.140,174.315,38.417,157.327
C08345=1057.228,382.164,384.180,174.310,38.410,157.326
C08346=1057.220,381.918,384.220,174.304,38.404,157.324
C08347=1057.213,381.671,384.261,174.299,38.397,157.322
C08348=1057.205,381.425,384.301,174.292,38.391,157.321
C08349=1057.197,381.178,384.342,174.287,38.384,157.319
C08350=1057.190,380.931,384.382,174.282,38.378,157.317
C08351=1057.182,380.685,384.423,174.276,38.371,157.315
C08352=1057.175,380.439,384.462,174.271,38.365,157.314
C08353=1057.168,380.192,384.503,174.265,38.359,157.312
C08354=1057.160,379.945,384.543,174.259,38.352,157.311
C08355=1057.153,379.698,384.583,174.254,38.346,157.309
C08356=1057.145,379.452,384.624,174.248,38.340,157.307
C08357=1057.137,379.205,384.664,174.243,38.334,157.306
C08358=1057.130,378.959,384.703,174.238,38.328,157.304
C08359=1057.122,378.712,384.743,174.232,38.321,157.302
C08360=1057.114,378.466,384.784,174.226,38.315,157.301
C08361=1057.106,378.219,384.824,174.220,38.309,157.299
C08362=1057.099,377.973,384.863,174.215,38.303,157.298
C08363=1057.091,377.726,384.903,174.210,38.296,157.296
C08364=1057.084,377.479,384.943,174.205,38.290,157.295
C08365=1057.077,377.233,384.983,174.199,38.284,157.293
C08366=1057.069,376.986,385.023,174.194,38.278,157.291
C08367=1057.061,376.739,385.063,174.188,38.271,157.290
C08368=1057.054,376.493,385.102,174.183,38.265,157.288
C08369=1057.046,376.246,385.142,174.178,38.259,157.287
C08370=1057.039,375.999,385.182,174.173,38.253,157.285
C08371=1057.031,375.753,385.222,174.166,38.247,157.283
C08372=1057.024,375.506,385.262,174.161,38.241,157.282
C08373=1057.017,375.260,385.301,174.156,38.235,157.280
C08374=1057.009,375.013,385.341,174.150,38.229,157.279
C08375=1057.001,374.765,385.380,174.145,38.223,157.277
C08376=1056.994,374.519,385.420,174.140,38.217,157.276
C08377=1056.986,374.236,385.465,174.134,38.210,157.274
C08378=1056.977,373.953,385.510,174.128,38.203,157.272
C08379=1056.969,373.671,385.556,174.122,38.196,157.270
C08380=1056.960,373.389,385.601,174.116,38.189,157.268
C08381=1056.953,373.142,385.640,174.111,38.183,157.267
C08382=1056.946,372.895,385.679,174.105,38.177,157.265
C08383=1056.938,372.648,385.719,174.100,38.171,157.264
C08384=1056.931,372.402,385.758,174.095,38.165,157.263
C08385=1056.923,372.155,385.798,174.090,38.159,157.261
C08386=1056.917,371.908,385.837,174.085,38.153,157.259
C08387=1056.909,371.661,385.877,174.079,38.147,157.258
C08388=1056.901,371.414,385.915,174.074,38.141,157.256
C08389=1056.894,371.168,385.954,174.069,38.136,157.255
C08390=1056.887,370.921,385.994,174.064,38.130,157.254
C08391=1056.879,370.674,386.032,174.059,38.124,157.252
C08392=1056.871,370.427,386.072,174.053,38.119,157.251
C08393=1056.864,370.181,386.110,174.048,38.113,157.249
C08394=1056.856,369.933,386.149,174.044,38.107,157.248
C08395=1056.850,369.686,386.188,174.039,38.101,157.246
C08396=1056.842,369.441,386.227,174.034,38.095,157.245
C08397=1056.834,369.193,386.266,174.028,38.090,157.243
C08398=1056.828,368.946,386.305,174.023,38.084,157.242
C08399=1056.820,368.700,386.344,174.018,38.078,157.240
C08400=1056.813,368.452,386.383,174.013,38.072,157.239
C08401=1056.805,368.206,386.421,174.008,38.067,157.237
C08402=1056.798,367.959,386.461,174.003,38.061,157.236
C08403=1056.791,367.713,386.499,173.997,38.055,157.235
C08404=1056.783,367.465,386.538,173.993,38.050,157.233
C08405=1056.776,367.219,386.577,173.988,38.044,157.232
C08406=1056.769,366.972,386.615,173.983,38.038,157.230
C08407=1056.762,366.725,386.654,173.978,38.033,157.229
C08408=1056.754,366.478,386.693,173.973,38.027,157.227
C08409=1056.747,366.231,386.731,173.968,38.021,157.226
C08410=1056.740,365.984,386.770,173.963,38.016,157.225
C08411=1056.733,365.737,386.808,173.958,38.010,157.223
C08412=1056.726,365.490,386.847,173.953,38.004,157.222
C08413=1056.718,365.243,386.885,173.948,37.999,157.220
C08414=1056.711,364.996,386.924,173.943,37.994,157.219
C08415=1056.704,364.750,386.963,173.939,37.988,157.218
C08416=1056.697,364.503,387.001,173.934,37.983,157.216
C08417=1056.690,364.256,387.039,173.929,37.976,157.215
C08418=1056.683,364.009,387.077,173.923,37.971,157.213
C08419=1056.676,363.762,387.116,173.918,37.966,157.212
C08420=1056.669,363.515,387.154,173.914,37.960,157.211
C08421=1056.662,363.268,387.193,173.909,37.955,157.209
C08422=1056.654,363.021,387.231,173.904,37.949,157.208
C08423=1056.646,362.774,387.269,173.899,37.944,157.207
C08424=1056.640,362.527,387.308,173.895,37.939,157.205
C08425=1056.632,362.280,387.345,173.890,37.933,157.204
C08426=1056.625,362.033,387.383,173.885,37.928,157.203
C08427=1056.617,361.786,387.421,173.880,37.922,157.201
C08428=1056.611,361.540,387.460,173.876,37.917,157.200
C08429=1056.603,361.292,387.497,173.871,37.911,157.198
C08430=1056.596,361.046,387.535,173.866,37.906,157.197
C08431=1056.589,360.798,387.574,173.861,37.901,157.196
C08432=1056.582,360.551,387.611,173.857,37.895,157.194
C08433=1056.574,360.287,387.652,173.851,37.890,157.193
C08434=1056.566,360.024,387.692,173.846,37.884,157.192
C08435=1056.558,359.759,387.733,173.841,37.878,157.190
C08436=1056.551,359.495,387.774,173.836,37.873,157.189
C08437=1056.544,359.248,387.811,173.831,37.867,157.187
C08438=1056.537,359.000,387.849,173.827,37.862,157.186
C08439=1056.530,358.753,387.887,173.822,37.857,157.185
C08440=1056.522,358.507,387.925,173.817,37.851,157.184
C08441=1056.515,358.260,387.962,173.813,37.846,157.182
C08442=1056.508,358.013,388.000,173.808,37.841,157.181
C08443=1056.502,357.766,388.038,173.803,37.836,157.180
C08444=1056.495,357.519,388.075,173.799,37.830,157.178
C08445=1056.488,357.272,388.113,173.794,37.825,157.177
C08446=1056.480,357.024,388.150,173.789,37.820,157.176
C08447=1056.473,356.777,388.188,173.785,37.815,157.175
C08448=1056.466,356.530,388.225,173.780,37.810,157.173
C08449=1056.459,356.283,388.263,173.775,37.804,157.172
C08450=1056.451,356.036,388.300,173.771,37.799,157.171
C08451=1056.445,355.789,388.338,173.766,37.794,157.169
C08452=1056.437,355.542,388.375,173.761,37.789,157.168
C08453=1056.430,355.295,388.413,173.757,37.784,157.167
C08454=1056.423,355.048,388.450,173.752,37.779,157.166
C08455=1056.416,354.800,388.487,173.748,37.774,157.164
C08456=1056.409,354.554,388.524,173.743,37.768,157.163
C08457=1056.402,354.307,388.562,173.738,37.763,157.162
C08458=1056.395,354.060,388.599,173.734,37.758,157.161
C08459=1056.388,353.812,388.637,173.729,37.754,157.159
C08460=1056.381,353.565,388.674,173.725,37.749,157.158
C08461=1056.374,353.318,388.711,173.721,37.744,157.157
C08462=1056.367,353.071,388.748,173.716,37.738,157.156
C08463=1056.360,352.823,388.785,173.712,37.733,157.154
C08464=1056.353,352.577,388.822,173.708,37.728,157.153
C08465=1056.346,352.330,388.860,173.703,37.723,157.152
C08466=1056.339,352.082,388.897,173.698,37.718,157.151
C08467=1056.332,351.836,388.934,173.694,37.713,157.150
C08468=1056.325,351.588,388.971,173.689,37.708,157.148
C08469=1056.318,351.341,389.008,173.685,37.703,157.147
C08470=1056.311,351.094,389.044,173.680,37.698,157.146
C08471=1056.304,350.847,389.081,173.676,37.693,157.145
C08472=1056.297,350.599,389.118,173.671,37.688,157.143
C08473=1056.290,350.353,389.155,173.667,37.683,157.142
C08474=1056.283,350.105,389.192,173.662,37.678,157.141
C08475=1056.275,349.858,389.229,173.659,37.674,157.140
C08476=1056.269,349.611,389.266,173.654,37.669,157.139
C08477=1056.262,349.363,389.302,173.650,37.664,157.137
C08478=1056.254,349.116,389.339,173.645,37.659,157.136
C08479=1056.248,348.869,389.376,173.641,37.654,157.135
C08480=1056.241,348.622,389.413,173.636,37.649,157.134
C08481=1056.235,348.375,389.449,173.632,37.644,157.133
C08482=1056.227,348.128,389.486,173.627,37.639,157.132
C08483=1056.220,347.881,389.522,173.623,37.634,157.130
C08484=1056.213,347.633,389.559,173.618,37.630,157.129
C08485=1056.206,347.385,389.596,173.615,37.625,157.128
C08486=1056.199,347.138,389.632,173.611,37.620,157.127
C08487=1056.192,346.891,389.669,173.606,37.615,157.126
C08488=1056.186,346.644,389.706,173.602,37.610,157.125
C08489=1056.178,346.385,389.744,173.597,37.605,157.123
C08490=1056.171,346.125,389.782,173.592,37.600,157.122
C08491=1056.163,345.866,389.820,173.588,37.595,157.121
C08492=1056.157,345.607,389.859,173.583,37.590,157.120
C08493=1056.150,345.360,389.894,173.579,37.585,157.118
C08494=1056.143,345.112,389.931,173.575,37.581,157.117
C08495=1056.136,344.865,389.967,173.571,37.576,157.116
C08496=1056.129,344.618,390.003,173.567,37.571,157.115
C08497=1056.122,344.370,390.040,173.562,37.566,157.114
C08498=1056.115,344.124,390.076,173.558,37.561,157.113
C08499=1056.108,343.876,390.113,173.554,37.557,157.112
C08500=1056.101,343.629,390.149,173.549,37.552,157.110
C08501=1056.095,343.382,390.185,173.546,37.547,157.109
C08502=1056.088,343.134,390.221,173.541,37.543,157.108
C08503=1056.081,342.887,390.257,173.537,37.538,157.107
C08504=1056.073,342.640,390.293,173.533,37.533,157.106
C08505=1056.067,342.393,390.330,173.528,37.529,157.105
C08506=1056.060,342.145,390.365,173.524,37.524,157.104
C08507=1056.053,341.897,390.402,173.521,37.519,157.103
C08508=1056.046,341.651,390.438,173.516,37.515,157.102
C08509=1056.039,341.403,390.473,173.512,37.510,157.100
C08510=1056.033,341.156,390.510,173.508,37.505,157.099
C08511=1056.026,340.909,390.545,173.503,37.501,157.098
C08512=1056.018,340.661,390.581,173.500,37.497,157.097
C08513=1056.012,340.414,390.617,173.495,37.491,157.096
C08514=1056.005,340.166,390.653,173.491,37.487,157.095
C08515=1055.998,339.920,390.688,173.487,37.483,157.094
C08516=1055.991,339.671,390.724,173.483,37.478,157.093
C08517=1055.984,339.424,390.760,173.479,37.474,157.092
C08518=1055.978,339.177,390.796,173.475,37.469,157.090
C08519=1055.971,338.929,390.832,173.471,37.464,157.089
C08520=1055.964,338.682,390.867,173.466,37.460,157.088
C08521=1055.957,338.435,390.904,173.462,37.455,157.087
C08522=1055.951,338.188,390.939,173.459,37.451,157.086
C08523=1055.944,337.940,390.974,173.454,37.446,157.085
C08524=1055.936,337.693,391.010,173.450,37.442,157.084
C08525=1055.930,337.445,391.046,173.446,37.437,157.083
C08526=1055.923,337.198,391.082,173.443,37.433,157.082
C08527=1055.916,336.951,391.117,173.438,37.428,157.081
C08528=1055.910,336.703,391.153,173.434,37.423,157.080
C08529=1055.903,336.455,391.188,173.430,37.419,157.079
C08530=1055.896,336.208,391.224,173.426,37.414,157.077
C08531=1055.889,335.961,391.259,173.422,37.410,157.076
C08532=1055.882,335.714,391.294,173.418,37.406,157.075
C08533=1055.876,335.466,391.330,173.414,37.401,157.074
C08534=1055.869,335.219,391.365,173.410,37.397,157.073
C08535=1055.862,334.971,391.401,173.406,37.392,157.072
C08536=1055.855,334.724,391.437,173.402,37.388,157.071
C08537=1055.848,334.477,391.472,173.398,37.383,157.070
C08538=1055.842,334.229,391.507,173.394,37.379,157.069
C08539=1055.835,333.982,391.542,173.390,37.375,157.068
C08540=1055.828,333.734,391.577,173.386,37.370,157.067
C08541=1055.821,333.487,391.612,173.382,37.366,157.066
C08542=1055.815,333.240,391.647,173.378,37.361,157.065
C08543=1055.808,332.992,391.683,173.375,37.357,157.064
C08544=1055.801,332.745,391.718,173.370,37.352,157.063
C08545=1055.794,332.481,391.755,173.366,37.348,157.062
C08546=1055.787,332.217,391.793,173.362,37.343,157.061
C08547=1055.780,331.954,391.830,173.358,37.339,157.060
C08548=1055.772,331.690,391.867,173.354,37.334,157.058
C08549=1055.766,331.443,391.903,173.350,37.330,157.057
C08550=1055.759,331.195,391.938,173.346,37.325,157.056
C08551=1055.752,330.948,391.973,173.342,37.321,157.055
C08552=1055.745,330.701,392.008,173.338,37.316,157.054
C08553=1055.738,330.453,392.043,173.334,37.312,157.053
C08554=1055.733,330.206,392.077,173.330,37.308,157.052
C08555=1055.725,329.958,392.113,173.327,37.303,157.051
C08556=1055.718,329.711,392.147,173.323,37.299,157.050
C08557=1055.711,329.463,392.182,173.318,37.295,157.049
C08558=1055.704,329.215,392.217,173.315,37.291,157.048
C08559=1055.697,328.968,392.251,173.311,37.287,157.047
C08560=1055.691,328.720,392.286,173.307,37.282,157.046
C08561=1055.684,328.473,392.321,173.304,37.278,157.045
C08562=1055.677,328.225,392.355,173.300,37.274,157.044
C08563=1055.670,327.978,392.390,173.296,37.270,157.043
C08564=1055.663,327.730,392.424,173.291,37.265,157.042
C08565=1055.656,327.483,392.459,173.288,37.262,157.041
C08566=1055.650,327.236,392.493,173.284,37.257,157.040
C08567=1055.643,326.988,392.528,173.280,37.253,157.039
C08568=1055.636,326.741,392.562,173.277,37.249,157.039
C08569=1055.629,326.493,392.597,173.273,37.245,157.037
C08570=1055.623,326.245,392.631,173.269,37.241,157.037
C08571=1055.615,325.998,392.666,173.266,37.236,157.035
C08572=1055.609,325.750,392.700,173.262,37.232,157.035
C08573=1055.602,325.503,392.735,173.257,37.228,157.034
C08574=1055.595,325.255,392.769,173.254,37.224,157.033
C08575=1055.589,325.008,392.803,173.250,37.220,157.032
C08576=1055.581,324.761,392.838,173.246,37.216,157.031
C08577=1055.575,324.513,392.872,173.243,37.211,157.030
C08578=1055.569,324.265,392.907,173.239,37.207,157.029
C08579=1055.561,324.017,392.941,173.235,37.203,157.028
C08580=1055.555,323.770,392.976,173.232,37.199,157.027
C08581=1055.548,323.523,393.009,173.228,37.195,157.026
C08582=1055.541,323.275,393.044,173.224,37.191,157.025
C08583=1055.535,323.027,393.078,173.221,37.187,157.024
C08584=1055.528,322.780,393.113,173.217,37.182,157.023
C08585=1055.522,322.533,393.147,173.213,37.178,157.022
C08586=1055.514,322.285,393.180,173.210,37.174,157.021
C08587=1055.508,322.037,393.215,173.206,37.170,157.020
C08588=1055.501,321.789,393.249,173.202,37.166,157.019
C08589=1055.495,321.542,393.283,173.199,37.162,157.018
C08590=1055.488,321.295,393.318,173.195,37.158,157.017
C08591=1055.481,321.047,393.352,173.191,37.154,157.016
C08592=1055.475,320.800,393.386,173.188,37.149,157.015
C08593=1055.468,320.552,393.420,173.184,37.145,157.014
C08594=1055.461,320.304,393.454,173.180,37.141,157.013
C08595=1055.455,320.057,393.487,173.177,37.137,157.013
C08596=1055.448,319.809,393.522,173.173,37.133,157.012
C08597=1055.441,319.561,393.556,173.169,37.129,157.011
C08598=1055.435,319.314,393.590,173.166,37.125,157.010
C08599=1055.429,319.066,393.624,173.162,37.121,157.009
C08600=1055.422,318.819,393.658,173.158,37.117,157.008
C08601=1055.415,318.550,393.695,173.155,37.112,157.007
C08602=1055.408,318.280,393.731,173.150,37.108,157.006
C08603=1055.401,318.012,393.768,173.146,37.104,157.005
C08604=1055.394,317.743,393.805,173.143,37.099,157.004
C08605=1055.388,317.496,393.839,173.139,37.095,157.003
C08606=1055.380,317.248,393.873,173.135,37.091,157.002
C08607=1055.375,317.001,393.907,173.132,37.087,157.001
C08608=1055.368,316.753,393.940,173.128,37.083,157.000
C08609=1055.362,316.505,393.974,173.125,37.079,156.999
C08610=1055.355,316.258,394.008,173.121,37.075,156.998
C08611=1055.349,316.010,394.042,173.117,37.071,156.997
C08612=1055.342,315.763,394.076,173.114,37.067,156.996
C08613=1055.336,315.515,394.109,173.111,37.063,156.995
C08614=1055.329,315.267,394.143,173.107,37.059,156.994
C08615=1055.323,315.020,394.177,173.104,37.055,156.994
C08616=1055.316,314.772,394.210,173.100,37.051,156.993
C08617=1055.310,314.524,394.244,173.097,37.047,156.992
C08618=1055.303,314.277,394.278,173.093,37.043,156.991
C08619=1055.297,314.029,394.311,173.089,37.038,156.990
C08620=1055.291,313.782,394.345,173.086,37.034,156.989
C08621=1055.284,313.534,394.378,173.082,37.030,156.988
C08622=1055.278,313.286,394.412,173.079,37.026,156.987
C08623=1055.271,313.038,394.446,173.076,37.023,156.986
C08624=1055.265,312.791,394.478,173.072,37.019,156.985
C08625=1055.258,312.543,394.511,173.069,37.015,156.984
C08626=1055.251,312.296,394.545,173.065,37.011,156.984
C08627=1055.244,312.047,394.578,173.062,37.007,156.983
C08628=1055.238,311.800,394.611,173.058,37.003,156.982
C08629=1055.231,311.552,394.645,173.054,36.999,156.981
C08630=1055.224,311.305,394.677,173.051,36.995,156.980
C08631=1055.216,311.057,394.711,173.047,36.992,156.979
C08632=1055.210,310.810,394.743,173.045,36.988,156.978
C08633=1055.204,310.562,394.776,173.041,36.984,156.977
C08634=1055.197,310.314,394.810,173.037,36.981,156.977
C08635=1055.190,310.067,394.843,173.034,36.977,156.976
C08636=1055.184,309.818,394.876,173.030,36.973,156.975
C08637=1055.177,309.571,394.909,173.027,36.968,156.974
C08638=1055.170,309.323,394.942,173.023,36.965,156.973
C08639=1055.164,309.075,394.975,173.020,36.961,156.972
C08640=1055.157,308.828,395.008,173.017,36.957,156.971
C08641=1055.151,308.580,395.041,173.013,36.954,156.970
C08642=1055.144,308.333,395.074,173.010,36.950,156.970
C08643=1055.137,308.085,395.106,173.006,36.946,156.969
C08644=1055.130,307.837,395.140,173.003,36.942,156.968
C08645=1055.124,307.589,395.172,172.999,36.938,156.967
C08646=1055.117,307.342,395.205,172.997,36.934,156.966
C08647=1055.111,307.094,395.238,172.993,36.931,156.965
C08648=1055.104,306.846,395.271,172.989,36.927,156.964
C08649=1055.098,306.598,395.304,172.986,36.923,156.963
C08650=1055.091,306.351,395.337,172.982,36.919,156.963
C08651=1055.084,306.103,395.370,172.979,36.915,156.962
C08652=1055.077,305.856,395.402,172.976,36.912,156.961
C08653=1055.071,305.608,395.435,172.973,36.908,156.960
C08654=1055.065,305.361,395.468,172.969,36.904,156.959
C08655=1055.059,305.113,395.501,172.966,36.900,156.958
C08656=1055.052,304.865,395.534,172.962,36.896,156.957
C08657=1055.045,304.600,395.568,172.958,36.892,156.957
C08658=1055.038,304.336,395.603,172.956,36.888,156.956
C08659=1055.030,304.071,395.638,172.952,36.884,156.955
C08660=1055.024,303.807,395.673,172.949,36.880,156.954
C08661=1055.017,303.559,395.705,172.945,36.876,156.953
C08662=1055.011,303.311,395.738,172.941,36.873,156.952
C08663=1055.005,303.063,395.770,172.938,36.869,156.951
C08664=1054.999,302.816,395.803,172.935,36.865,156.951
C08665=1054.992,302.567,395.836,172.932,36.861,156.950
C08666=1054.985,302.320,395.868,172.928,36.857,156.949
C08667=1054.978,302.072,395.901,172.925,36.854,156.948
C08668=1054.972,301.825,395.934,172.922,36.850,156.947
C08669=1054.966,301.577,395.966,172.919,36.846,156.946
C08670=1054.960,301.329,395.998,172.915,36.842,156.945
C08671=1054.954,301.081,396.031,172.912,36.839,156.945
C08672=1054.947,300.834,396.063,172.909,36.835,156.944
C08673=1054.941,300.586,396.095,172.905,36.831,156.943
C08674=1054.934,300.338,396.128,172.902,36.827,156.942
C08675=1054.927,300.090,396.161,172.899,36.823,156.941
C08676=1054.921,299.842,396.193,172.896,36.820,156.940
C08677=1054.914,299.594,396.225,172.892,36.816,156.939
C08678=1054.908,299.347,396.258,172.890,36.812,156.939
C08679=1054.902,299.099,396.290,172.886,36.808,156.938
C08680=1054.896,298.851,396.323,172.883,36.805,156.937
C08681=1054.890,298.603,396.355,172.880,36.801,156.936
C08682=1054.883,298.356,396.387,172.877,36.797,156.935
C08683=1054.876,298.108,396.420,172.873,36.793,156.934
C08684=1054.870,297.860,396.452,172.870,36.790,156.934
C08685=1054.864,297.612,396.485,172.867,36.786,156.933
C08686=1054.857,297.364,396.516,172.863,36.782,156.932
C08687=1054.852,297.117,396.548,172.861,36.778,156.931
C08688=1054.846,296.869,396.580,172.857,36.774,156.930
C08689=1054.840,296.622,396.613,172.854,36.771,156.929
C08690=1054.833,296.374,396.645,172.851,36.767,156.929
C08691=1054.827,296.125,396.677,172.848,36.763,156.928
C08692=1054.820,295.878,396.709,172.844,36.760,156.927
C08693=1054.814,295.630,396.741,172.842,36.756,156.926
C08694=1054.807,295.382,396.772,172.838,36.752,156.925
C08695=1054.801,295.134,396.805,172.835,36.749,156.924
C08696=1054.794,294.887,396.836,172.832,36.745,156.924
C08697=1054.788,294.638,396.868,172.829,36.741,156.923
C08698=1054.781,294.391,396.901,172.825,36.738,156.922
C08699=1054.774,294.143,396.932,172.823,36.734,156.921
C08700=1054.768,293.895,396.964,172.819,36.730,156.920
C08701=1054.762,293.647,396.995,172.816,36.727,156.920
C08702=1054.756,293.399,397.027,172.813,36.723,156.919
C08703=1054.749,293.152,397.060,172.810,36.719,156.918
C08704=1054.742,292.904,397.091,172.807,36.716,156.917
C08705=1054.736,292.655,397.123,172.804,36.712,156.916
C08706=1054.729,292.408,397.154,172.800,36.709,156.916
C08707=1054.722,292.160,397.186,172.798,36.705,156.915
C08708=1054.716,291.911,397.218,172.794,36.701,156.914
C08709=1054.710,291.664,397.249,172.792,36.698,156.913
C08710=1054.703,291.417,397.281,172.788,36.694,156.912
C08711=1054.697,291.169,397.313,172.785,36.690,156.912
C08712=1054.691,290.921,397.345,172.782,36.687,156.911
C08713=1054.684,290.671,397.376,172.779,36.683,156.910
C08714=1054.678,290.423,397.408,172.776,36.679,156.909
C08715=1054.671,290.174,397.439,172.773,36.676,156.908
C08716=1054.665,289.926,397.471,172.769,36.672,156.908
C08717=1054.659,289.678,397.503,172.767,36.669,156.907
C08718=1054.652,289.430,397.534,172.763,36.665,156.906
C08719=1054.645,289.182,397.566,172.761,36.661,156.905
C08720=1054.639,288.934,397.598,172.757,36.658,156.904
C08721=1054.632,288.686,397.629,172.754,36.654,156.904
C08722=1054.627,288.438,397.660,172.751,36.651,156.903
C08723=1054.620,288.190,397.691,172.748,36.647,156.902
C08724=1054.613,287.942,397.722,172.745,36.643,156.901
C08725=1054.607,287.694,397.754,172.742,36.640,156.900
C08726=1054.600,287.446,397.786,172.739,36.636,156.900
C08727=1054.594,287.198,397.817,172.736,36.633,156.899
C08728=1054.588,286.950,397.848,172.733,36.629,156.898
C08729=1054.581,286.702,397.879,172.730,36.626,156.897
C08730=1054.574,286.455,397.911,172.726,36.622,156.897
C08731=1054.568,286.207,397.942,172.724,36.619,156.896
C08732=1054.561,285.958,397.973,172.720,36.615,156.895
C08733=1054.555,285.711,398.004,172.718,36.611,156.894
C08734=1054.548,285.463,398.035,172.714,36.608,156.893
C08735=1054.542,285.214,398.066,172.712,36.604,156.893
C08736=1054.535,284.967,398.097,172.709,36.601,156.892
C08737=1054.529,284.719,398.128,172.706,36.597,156.891
C08738=1054.523,284.471,398.159,172.703,36.594,156.890
C08739=1054.516,284.223,398.191,172.700,36.590,156.890
C08740=1054.509,283.975,398.222,172.697,36.587,156.889
C08741=1054.503,283.727,398.252,172.694,36.583,156.888
C08742=1054.497,283.479,398.284,172.691,36.579,156.887
C08743=1054.490,283.231,398.314,172.688,36.576,156.886
C08744=1054.484,282.984,398.346,172.685,36.572,156.886
C08745=1054.477,282.736,398.377,172.682,36.569,156.885
C08746=1054.471,282.487,398.408,172.679,36.565,156.884
C08747=1054.465,282.240,398.439,172.676,36.562,156.883
C08748=1054.459,281.991,398.469,172.673,36.558,156.883
C08749=1054.452,281.744,398.501,172.670,36.555,156.882
C08750=1054.446,281.496,398.531,172.667,36.551,156.881
C08751=1054.439,281.248,398.563,172.665,36.548,156.880
C08752=1054.433,280.999,398.593,172.661,36.544,156.879
C08753=1054.427,280.751,398.624,172.659,36.540,156.879
C08754=1054.420,280.504,398.655,172.656,36.537,156.878
C08755=1054.414,280.256,398.686,172.653,36.533,156.877
C08756=1054.408,280.008,398.717,172.650,36.530,156.876
C08757=1054.401,279.759,398.748,172.647,36.526,156.876
C08758=1054.396,279.511,398.778,172.644,36.523,156.875
C08759=1054.389,279.264,398.809,172.641,36.519,156.874
C08760=1054.382,279.015,398.840,172.638,36.516,156.873
C08761=1054.377,278.767,398.871,172.635,36.512,156.873
C08762=1054.369,278.520,398.901,172.632,36.509,156.872
C08763=1054.363,278.272,398.932,172.630,36.505,156.871
C08764=1054.357,278.023,398.962,172.627,36.501,156.870
C08765=1054.350,277.780,398.993,172.624,36.498,156.869
C08766=1054.345,277.538,399.022,172.621,36.494,156.869
C08767=1054.337,277.295,399.052,172.618,36.492,156.868
C08768=1054.332,277.052,399.082,172.616,36.488,156.867
C08769=1054.325,276.809,399.112,172.612,36.485,156.867
C08770=1054.319,276.567,399.142,172.610,36.481,156.866
C08771=1054.313,276.324,399.172,172.607,36.478,156.865
C08772=1054.307,276.081,399.202,172.604,36.474,156.864
C08773=1054.300,275.833,399.232,172.602,36.470,156.864
C08774=1054.294,275.585,399.262,172.598,36.467,156.863
C08775=1054.288,275.337,399.293,172.596,36.463,156.862
C08776=1054.281,275.089,399.323,172.593,36.460,156.861
C08777=1054.275,274.841,399.354,172.590,36.456,156.860
C08778=1054.268,274.592,399.384,172.587,36.453,156.860
C08779=1054.263,274.344,399.415,172.584,36.450,156.859
C08780=1054.255,274.096,399.445,172.582,36.446,156.858
C08781=1054.250,273.848,399.475,172.579,36.443,156.858
C08782=1054.243,273.600,399.506,172.576,36.439,156.857
C08783=1054.237,273.352,399.536,172.573,36.436,156.856
C08784=1054.231,273.104,399.566,172.571,36.432,156.855
C08785=1054.224,272.856,399.596,172.567,36.429,156.855
C08786=1054.218,272.608,399.627,172.565,36.425,156.854
C08787=1054.211,272.360,399.657,172.561,36.422,156.853
C08788=1054.205,272.112,399.687,172.559,36.418,156.852
C08789=1054.198,271.864,399.718,172.557,36.415,156.852
C08790=1054.192,271.616,399.747,172.553,36.411,156.851
C08791=1054.185,271.368,399.778,172.551,36.408,156.850
C08792=1054.179,271.120,399.807,172.548,36.404,156.849
C08793=1054.173,270.871,399.838,172.545,36.401,156.849
C08794=1054.166,270.623,399.868,172.542,36.398,156.848
C08795=1054.160,270.375,399.898,172.540,36.394,156.847
C08796=1054.153,270.127,399.928,172.537,36.391,156.846
C08797=1054.148,269.879,399.958,172.534,36.387,156.846
C08798=1054.141,269.631,399.988,172.532,36.384,156.845
C08799=1054.135,269.383,400.018,172.528,36.380,156.844
C08800=1054.128,269.135,400.048,172.526,36.377,156.843
C08801=1054.122,268.886,400.078,172.523,36.373,156.843
C08802=1054.116,268.639,400.108,172.520,36.370,156.842
C08803=1054.109,268.390,400.139,172.518,36.367,156.841
C08804=1054.103,268.142,400.168,172.515,36.363,156.840
C08805=1054.096,267.894,400.198,172.512,36.360,156.840
C08806=1054.090,267.646,400.228,172.509,36.356,156.839
C08807=1054.084,267.398,400.257,172.507,36.353,156.838
C08808=1054.077,267.149,400.288,172.504,36.349,156.837
C08809=1054.071,266.901,400.317,172.501,36.346,156.837
C08810=1054.064,266.654,400.347,172.499,36.343,156.836
C08811=1054.058,266.405,400.377,172.496,36.339,156.835
C08812=1054.052,266.157,400.406,172.493,36.336,156.835
C08813=1054.045,265.909,400.436,172.490,36.332,156.834
C08814=1054.039,265.660,400.466,172.488,36.328,156.833
C08815=1054.033,265.413,400.496,172.485,36.325,156.832
C08816=1054.026,265.165,400.525,172.482,36.322,156.832
C08817=1054.020,264.916,400.556,172.480,36.318,156.831
C08818=1054.014,264.668,400.585,172.477,36.315,156.830
C08819=1054.007,264.421,400.614,172.474,36.311,156.829
C08820=1054.001,264.172,400.644,172.471,36.308,156.829
C08821=1053.995,263.931,400.672,172.469,36.304,156.828
C08822=1053.989,263.690,400.702,172.467,36.301,156.827
C08823=1053.983,263.450,400.730,172.464,36.298,156.827
C08824=1053.976,263.209,400.759,172.461,36.294,156.826
C08825=1053.970,262.968,400.788,172.458,36.291,156.825
C08826=1053.964,262.727,400.816,172.456,36.288,156.824
C08827=1053.957,262.486,400.845,172.454,36.285,156.824
C08828=1053.951,262.245,400.874,172.451,36.281,156.823
C08829=1053.945,261.997,400.903,172.448,36.278,156.822
C08830=1053.939,261.749,400.932,172.445,36.275,156.822
C08831=1053.932,261.500,400.962,172.443,36.271,156.821
C08832=1053.925,261.253,400.991,172.441,36.268,156.820
C08833=1053.919,261.005,401.020,172.437,36.265,156.820
C08834=1053.912,260.756,401.050,172.435,36.261,156.819
C08835=1053.906,260.508,401.079,172.432,36.258,156.818
C08836=1053.899,260.260,401.107,172.430,36.254,156.817
C08837=1053.892,260.012,401.137,172.427,36.251,156.817
C08838=1053.886,259.764,401.166,172.424,36.248,156.816
C08839=1053.879,259.515,401.195,172.422,36.244,156.815
C08840=1053.873,259.267,401.225,172.420,36.241,156.815
C08841=1053.867,259.019,401.254,172.417,36.238,156.814
C08842=1053.860,258.770,401.283,172.414,36.234,156.813
C08843=1053.854,258.522,401.312,172.411,36.231,156.812
C08844=1053.847,258.274,401.341,172.409,36.228,156.812
C08845=1053.841,258.027,401.371,172.406,36.224,156.811
C08846=1053.834,257.778,401.400,172.403,36.220,156.810
C08847=1053.828,257.530,401.429,172.401,36.218,156.810
C08848=1053.822,257.281,401.458,172.398,36.214,156.809
C08849=1053.815,257.033,401.487,172.396,36.210,156.808
C08850=1053.809,256.785,401.516,172.394,36.207,156.807
C08851=1053.803,256.537,401.545,172.391,36.204,156.807
C08852=1053.796,256.288,401.575,172.388,36.200,156.806
C08853=1053.790,256.040,401.604,172.385,36.197,156.805
C08854=1053.783,255.792,401.632,172.383,36.193,156.804
C08855=1053.776,255.544,401.661,172.381,36.190,156.804
C08856=1053.770,255.296,401.690,172.378,36.187,156.803
C08857=1053.764,255.047,401.719,172.375,36.183,156.802
C08858=1053.758,254.799,401.748,172.372,36.180,156.802
C08859=1053.751,254.550,401.777,172.370,36.177,156.801
C08860=1053.745,254.302,401.806,172.368,36.173,156.800
C08861=1053.739,254.054,401.835,172.365,36.170,156.799
C08862=1053.732,253.806,401.864,172.363,36.166,156.799
C08863=1053.726,253.558,401.893,172.360,36.163,156.798
C08864=1053.720,253.310,401.922,172.357,36.160,156.797
C08865=1053.713,253.061,401.950,172.355,36.156,156.797
C08866=1053.707,252.813,401.979,172.352,36.152,156.796
C08867=1053.701,252.565,402.008,172.350,36.149,156.795
C08868=1053.694,252.317,402.037,172.348,36.146,156.794
C08869=1053.688,252.069,402.066,172.345,36.142,156.794
C08870=1053.682,251.820,402.095,172.343,36.139,156.793
C08871=1053.676,251.572,402.124,172.340,36.135,156.792
C08872=1053.669,251.323,402.153,172.337,36.132,156.791
C08873=1053.663,251.075,402.182,172.335,36.129,156.791
C08874=1053.656,250.826,402.210,172.332,36.125,156.790
C08875=1053.650,250.578,402.239,172.330,36.122,156.789
C08876=1053.644,250.330,402.268,172.327,36.118,156.789
C08877=1053.638,250.088,402.296,172.325,36.115,156.788
C08878=1053.632,249.847,402.323,172.323,36.112,156.787
C08879=1053.626,249.606,402.352,172.320,36.108,156.787
C08880=1053.620,249.364,402.380,172.318,36.105,156.786
C08881=1053.614,249.122,402.407,172.316,36.101,156.785
C08882=1053.608,248.880,402.435,172.313,36.098,156.784
C08883=1053.601,248.638,402.463,172.311,36.094,156.784
C08884=1053.596,248.396,402.491,172.308,36.091,156.783
C08885=1053.590,248.148,402.520,172.306,36.088,156.782
C08886=1053.583,247.900,402.548,172.304,36.084,156.782
C08887=1053.577,247.652,402.577,172.301,36.081,156.781
C08888=1053.570,247.403,402.606,172.299,36.077,156.780
C08889=1053.564,247.155,402.634,172.296,36.074,156.779
C08890=1053.559,246.907,402.663,172.294,36.071,156.779
C08891=1053.553,246.658,402.691,172.291,36.067,156.778
C08892=1053.546,246.411,402.720,172.288,36.063,156.777
C08893=1053.540,246.162,402.748,172.286,36.060,156.776
C08894=1053.534,245.914,402.777,172.284,36.056,156.776
C08895=1053.528,245.665,402.805,172.281,36.053,156.775
C08896=1053.521,245.417,402.834,172.279,36.050,156.774
C08897=1053.515,245.168,402.862,172.276,36.046,156.774
C08898=1053.508,244.920,402.890,172.274,36.043,156.773
C08899=1053.502,244.672,402.919,172.272,36.040,156.772
C08900=1053.496,244.423,402.947,172.269,36.036,156.772
C08901=1053.489,244.175,402.976,172.267,36.033,156.771
C08902=1053.484,243.927,403.004,172.265,36.029,156.770
C08903=1053.477,243.679,403.031,172.262,36.025,156.769
C08904=1053.471,243.431,403.060,172.260,36.022,156.769
C08905=1053.465,243.182,403.089,172.257,36.019,156.768
C08906=1053.458,242.933,403.117,172.255,36.015,156.767
C08907=1053.452,242.685,403.145,172.253,36.012,156.766
C08908=1053.445,242.437,403.173,172.250,36.009,156.766
C08909=1053.439,242.188,403.202,172.248,36.005,156.765
C08910=1053.433,241.940,403.229,172.246,36.002,156.764
C08911=1053.427,241.692,403.258,172.243,35.998,156.764
C08912=1053.420,241.444,403.286,172.241,35.995,156.763
C08913=1053.414,241.195,403.314,172.238,35.991,156.762
C08914=1053.408,240.947,403.342,172.236,35.988,156.762
C08915=1053.401,240.698,403.370,172.234,35.984,156.761
C08916=1053.395,240.449,403.398,172.231,35.981,156.760
C08917=1053.388,240.202,403.426,172.229,35.978,156.759
C08918=1053.382,239.954,403.454,172.227,35.974,156.759
C08919=1053.376,239.705,403.482,172.224,35.971,156.758
C08920=1053.369,239.457,403.510,172.222,35.968,156.757
C08921=1053.363,239.208,403.538,172.220,35.964,156.757
C08922=1053.357,238.959,403.566,172.217,35.961,156.756
C08923=1053.350,238.711,403.594,172.215,35.958,156.755
C08924=1053.345,238.463,403.621,172.212,35.954,156.755
C08925=1053.338,238.215,403.649,172.210,35.950,156.754
C08926=1053.331,237.966,403.677,172.208,35.947,156.753
C08927=1053.325,237.718,403.705,172.205,35.944,156.752
C08928=1053.319,237.469,403.733,172.203,35.940,156.752
C08929=1053.313,237.221,403.760,172.201,35.937,156.751
C08930=1053.306,236.973,403.788,172.198,35.934,156.750
C08931=1053.299,236.724,403.816,172.196,35.930,156.750
C08932=1053.293,236.476,403.844,172.194,35.927,156.749
C08933=1053.287,236.231,403.872,172.191,35.923,156.748
C08934=1053.281,235.986,403.899,172.189,35.920,156.748
C08935=1053.274,235.741,403.927,172.188,35.916,156.747
C08936=1053.268,235.498,403.953,172.185,35.913,156.746
C08937=1053.262,235.253,403.981,172.183,35.910,156.745
C08938=1053.256,235.008,404.008,172.181,35.906,156.745
C08939=1053.250,234.763,404.035,172.178,35.903,156.744
C08940=1053.243,234.518,404.062,172.176,35.900,156.743
C08941=1053.237,234.270,404.090,172.173,35.896,156.743
C08942=1053.231,234.021,404.118,172.171,35.892,156.742
C08943=1053.225,233.773,404.146,172.169,35.889,156.741
C08944=1053.218,233.525,404.173,172.166,35.885,156.740
C08945=1053.211,233.276,404.201,172.164,35.882,156.740
C08946=1053.206,233.028,404.228,172.163,35.879,156.739
C08947=1053.200,232.779,404.256,172.160,35.875,156.738
C08948=1053.193,232.531,404.284,172.158,35.872,156.738
C08949=1053.187,232.283,404.311,172.156,35.868,156.737
C08950=1053.181,232.034,404.338,172.153,35.865,156.736
C08951=1053.174,231.785,404.366,172.151,35.861,156.735
C08952=1053.167,231.537,404.394,172.149,35.858,156.735
C08953=1053.162,231.289,404.422,172.146,35.854,156.734
C08954=1053.155,231.040,404.449,172.144,35.851,156.733
C08955=1053.149,230.792,404.476,172.142,35.848,156.733
C08956=1053.143,230.544,404.504,172.140,35.844,156.732
C08957=1053.136,230.295,404.531,172.138,35.841,156.731
C08958=1053.130,230.047,404.558,172.135,35.838,156.731
C08959=1053.124,229.798,404.586,172.133,35.834,156.730
C08960=1053.117,229.549,404.613,172.131,35.830,156.729
C08961=1053.111,229.302,404.640,172.128,35.827,156.728
C08962=1053.105,229.053,404.667,172.126,35.823,156.728
C08963=1053.098,228.804,404.695,172.124,35.820,156.727
C08964=1053.092,228.556,404.722,172.122,35.817,156.726
C08965=1053.086,228.307,404.749,172.120,35.813,156.726
C08966=1053.079,228.059,404.777,172.118,35.809,156.725
C08967=1053.073,227.811,404.804,172.115,35.806,156.724
C08968=1053.066,227.562,404.831,172.113,35.803,156.723
C08969=1053.060,227.313,404.858,172.111,35.799,156.723
C08970=1053.053,227.066,404.885,172.108,35.796,156.722
C08971=1053.047,226.817,404.912,172.107,35.793,156.721
C08972=1053.041,226.568,404.939,172.105,35.789,156.721
C08973=1053.034,226.320,404.967,172.102,35.785,156.720
C08974=1053.028,226.071,404.994,172.100,35.782,156.719
C08975=1053.022,225.823,405.021,172.098,35.779,156.719
C08976=1053.016,225.574,405.048,172.095,35.775,156.718
C08977=1053.005,225.180,405.090,172.092,35.770,156.717
C08978=1052.995,224.785,405.134,172.088,35.764,156.716
C08979=1052.985,224.390,405.177,172.086,35.758,156.714
C08980=1052.975,223.995,405.220,172.082,35.753,156.713
C08981=1052.969,223.747,405.247,172.080,35.750,156.713
C08982=1052.962,223.498,405.273,172.077,35.746,156.712
C08983=1052.956,223.250,405.301,172.075,35.743,156.711
C08984=1052.950,223.001,405.328,172.073,35.739,156.711
C08985=1052.944,222.753,405.354,172.071,35.736,156.710
C08986=1052.937,222.504,405.382,172.069,35.732,156.709
C08987=1052.932,222.256,405.409,172.067,35.729,156.708
C08988=1052.924,222.007,405.435,172.064,35.726,156.708
C08989=1052.916,221.657,405.473,172.062,35.720,156.707
C08990=1052.907,221.306,405.512,172.058,35.715,156.706
C08991=1052.898,220.954,405.549,172.056,35.711,156.705
C08992=1052.889,220.604,405.587,172.053,35.706,156.704
C08993=1052.883,220.356,405.614,172.050,35.702,156.703
C08994=1052.877,220.107,405.641,172.049,35.699,156.702
C08995=1052.870,219.858,405.667,172.046,35.695,156.702
C08996=1052.863,219.610,405.694,172.044,35.692,156.701
C08997=1052.858,219.362,405.721,172.042,35.688,156.700
C08998=1052.850,219.113,405.747,172.041,35.685,156.699
C08999=1052.845,218.865,405.774,172.038,35.681,156.699
C09000=1052.838,218.616,405.800,172.036,35.678,156.698
C09001=1052.832,218.367,405.827,172.034,35.674,156.697
C09002=1052.825,218.119,405.853,172.031,35.671,156.697
C09003=1052.819,217.870,405.880,172.030,35.667,156.696
C09004=1052.813,217.622,405.907,172.028,35.664,156.695
C09005=1052.806,217.373,405.933,172.025,35.660,156.694
C09006=1052.800,217.125,405.960,172.023,35.657,156.694
C09007=1052.793,216.876,405.986,172.022,35.653,156.693
C09008=1052.787,216.628,406.013,172.019,35.650,156.692
C09009=1052.781,216.380,406.039,172.017,35.646,156.692
C09010=1052.775,216.131,406.066,172.016,35.643,156.691
C09011=1052.769,215.882,406.093,172.013,35.639,156.690
C09012=1052.762,215.634,406.119,172.011,35.635,156.690
C09013=1052.756,215.385,406.146,172.009,35.632,156.689
C09014=1052.749,215.137,406.172,172.007,35.629,156.688
C09015=1052.743,214.888,406.199,172.005,35.625,156.687
C09016=1052.736,214.640,406.225,172.003,35.622,156.687
C09017=1052.730,214.391,406.252,172.000,35.618,156.686
C09018=1052.724,214.143,406.278,171.999,35.614,156.685
C09019=1052.718,213.895,406.305,171.997,35.611,156.685
C09020=1052.711,213.645,406.330,171.994,35.607,156.684
C09021=1052.705,213.397,406.357,171.993,35.604,156.683
C09022=1052.699,213.148,406.384,171.991,35.601,156.682
C09023=1052.692,212.900,406.410,171.988,35.597,156.682
C09024=1052.687,212.651,406.437,171.987,35.593,156.681
C09025=1052.680,212.403,406.463,171.985,35.590,156.680
C09026=1052.674,212.154,406.489,171.982,35.586,156.680
C09027=1052.667,211.906,406.515,171.980,35.583,156.679
C09028=1052.661,211.658,406.541,171.979,35.579,156.678
C09029=1052.655,211.408,406.568,171.976,35.575,156.677
C09030=1052.648,211.160,406.594,171.974,35.572,156.677
C09031=1052.642,210.912,406.620,171.973,35.569,156.676
C09032=1052.635,210.663,406.647,171.970,35.565,156.675
C09033=1052.629,210.415,406.673,171.968,35.561,156.675
C09034=1052.623,210.166,406.699,171.967,35.558,156.674
C09035=1052.617,209.918,406.725,171.964,35.554,156.673
C09036=1052.610,209.669,406.751,171.962,35.551,156.672
C09037=1052.604,209.420,406.776,171.961,35.547,156.672
C09038=1052.598,209.172,406.803,171.958,35.543,156.671
C09039=1052.591,208.923,406.829,171.956,35.540,156.670
C09040=1052.585,208.674,406.855,171.955,35.537,156.670
C09041=1052.579,208.428,406.881,171.953,35.533,156.669
C09042=1052.572,208.183,406.907,171.950,35.530,156.668
C09043=1052.565,207.937,406.933,171.949,35.526,156.667
C09044=1052.560,207.691,406.959,171.947,35.522,156.667
C09045=1052.553,207.445,406.984,171.945,35.519,156.666
C09046=1052.547,207.200,407.010,171.943,35.516,156.665
C09047=1052.540,206.953,407.035,171.941,35.512,156.665
C09048=1052.534,206.707,407.062,171.939,35.508,156.664
C09049=1052.509,205.656,407.167,171.720,35.414,156.647
C09050=1052.503,205.407,407.192,171.718,35.411,156.647
C09051=1052.496,205.158,407.216,171.716,35.409,156.646
C09052=1052.490,204.909,407.241,171.714,35.406,156.646
C09053=1052.485,204.661,407.266,171.710,35.403,156.645
C09054=1052.479,204.412,407.291,171.708,35.401,156.645
C09055=1052.473,204.163,407.316,171.706,35.398,156.644
C09056=1052.466,203.915,407.342,171.704,35.395,156.644
C09057=1052.461,203.666,407.366,171.701,35.392,156.643
C09058=1052.455,203.417,407.391,171.698,35.390,156.642
C09059=1052.449,203.168,407.416,171.696,35.387,156.642
C09060=1052.443,202.920,407.441,171.693,35.384,156.641
C09061=1052.437,202.671,407.465,171.691,35.381,156.641
C09062=1052.431,202.423,407.490,171.688,35.379,156.640
C09063=1052.425,202.174,407.514,171.686,35.376,156.640
C09064=1052.419,201.925,407.540,171.683,35.373,156.639
C09065=1052.413,201.676,407.564,171.681,35.371,156.639
C09066=1052.407,201.428,407.589,171.679,35.368,156.638
C09067=1052.401,201.179,407.613,171.676,35.365,156.638
C09068=1052.395,200.930,407.639,171.673,35.363,156.637
C09069=1052.388,200.681,407.663,171.671,35.360,156.637
C09070=1052.382,200.433,407.688,171.669,35.357,156.636
C09071=1052.377,200.184,407.712,171.667,35.355,156.636
C09072=1052.370,199.935,407.736,171.663,35.352,156.635
C09073=1052.364,199.687,407.761,171.661,35.350,156.635
C09074=1052.358,199.438,407.785,171.659,35.347,156.634
C09075=1052.352,199.189,407.810,171.657,35.344,156.634
C09076=1052.346,198.941,407.835,171.654,35.342,156.633
C09077=1052.339,198.692,407.859,171.651,35.339,156.633
C09078=1052.334,198.443,407.884,171.649,35.337,156.632
C09079=1052.327,198.195,407.908,171.647,35.334,156.632
C09080=1052.321,197.946,407.933,171.645,35.331,156.631
C09081=1052.315,197.697,407.957,171.642,35.329,156.631
C09082=1052.309,197.448,407.981,171.639,35.326,156.630
C09083=1052.303,197.200,408.006,171.637,35.324,156.630
C09084=1052.297,196.951,408.030,171.635,35.321,156.629
C09085=1052.291,196.702,408.054,171.632,35.318,156.629
C09086=1052.285,196.453,408.078,171.630,35.316,156.628
C09087=1052.279,196.205,408.103,171.627,35.313,156.628
C09088=1052.272,195.956,408.127,171.625,35.311,156.627
C09089=1052.267,195.707,408.152,171.623,35.308,156.627
C09090=1052.260,195.459,408.176,171.620,35.305,156.626
C09091=1052.255,195.209,408.200,171.618,35.303,156.626
C09092=1052.249,194.961,408.225,171.615,35.300,156.625
C09093=1052.242,194.712,408.249,171.613,35.298,156.625
C09094=1052.237,194.464,408.274,171.611,35.295,156.624
C09095=1052.230,194.215,408.298,171.608,35.292,156.624
C09096=1052.225,193.966,408.322,171.606,35.290,156.623
C09097=1052.218,193.717,408.346,171.603,35.287,156.623
C09098=1052.213,193.469,408.370,171.601,35.285,156.622
C09099=1052.206,193.220,408.394,171.599,35.283,156.622
C09100=1052.201,192.971,408.418,171.597,35.279,156.621
C09101=1052.195,192.722,408.443,171.594,35.277,156.621
C09102=1052.189,192.473,408.467,171.591,35.274,156.620
C09103=1052.183,192.224,408.491,171.589,35.272,156.620
C09104=1052.177,191.976,408.516,171.587,35.270,156.620
C09105=1052.170,191.728,408.540,171.585,35.267,156.619
C09106=1052.165,191.479,408.564,171.583,35.265,156.619
